QRS_NEXT_CUT()
PTP {E1 23936.911,E2 23936.911}
PTP {X 0,Y 607.929,A -85,B 0,C 180,E1 23936.911,E2 23936.911,E3 0,E4 0,E5 0,E6 0}
QRS_SPEED_INIT()
LIN {X 0,Y 607.929,Z 1180,A -85,B 0,C 180,E1 23936.911,E2 23936.911,E3 0,E4 0,E5 0,E6 0} C_VEL
LIN {X 0,Y 607.929,Z 517.391,A -85,B 0,C 180,E1 23936.911,E2 23936.911} C_VEL
LIN {X 0,Y 607.929,Z 509.316,A -85,B 0,C 180,E1 23936.911,E2 23936.911} C_VEL
LIN {X 0,Y 607.912,Z 507.316,A -85,B 0,C 180,E1 23936.722,E2 23936.722} C_VEL
LIN {X 0,Y 607.897,Z 507.324,A -85,B 0,C 180,E1 23933.441,E2 23933.441} C_VEL
LIN {X 0,Y 607.905,Z 507.318,A -85,B 0,C 180,E1 23930.246,E2 23930.246} C_VEL
LIN {X 0,Y 607.895,Z 507.323,A -85,B 0,C 180,E1 23927.074,E2 23927.074} C_VEL
LIN {X 0,Y 607.904,Z 507.318,A -85,B 0,C 180,E1 23923.861,E2 23923.861} C_VEL
LIN {X 0,Y 607.891,Z 507.323,A -85,B 0,C 180,E1 23920.694,E2 23920.694} C_VEL
LIN {X 0,Y 607.905,Z 507.318,A -85,B 0,C 180,E1 23917.568,E2 23917.568} C_VEL
LIN {X 0,Y 607.89,Z 507.323,A -85,B 0,C 180,E1 23914.337,E2 23914.337} C_VEL
LIN {X 0,Y 607.906,Z 507.318,A -85,B 0,C 180,E1 23911.189,E2 23911.189} C_VEL
LIN {X 0,Y 607.89,Z 507.324,A -85,B 0,C 180,E1 23908.02,E2 23908.02} C_VEL
LIN {X 0,Y 607.906,Z 507.318,A -85,B 0,C 180,E1 23904.83,E2 23904.83} C_VEL
LIN {X 0,Y 607.889,Z 507.324,A -85,B 0,C 180,E1 23901.677,E2 23901.677} C_VEL
LIN {X 0,Y 607.912,Z 507.317,A -85,B 0,C 180,E1 23898.591,E2 23898.591} C_VEL
LIN {X 0,Y 607.89,Z 507.324,A -85,B 0,C 180,E1 23895.386,E2 23895.386} C_VEL
LIN {X 0,Y 607.912,Z 507.315,A -85,B 0,C 180,E1 23892.257,E2 23892.257} C_VEL
LIN {X 0,Y 607.889,Z 507.318,A -85,B 0,C 180,E1 23889.047,E2 23889.047} C_VEL
LIN {X 0,Y 607.907,Z 507.606,A -85,B 0,C 180,E1 23887.52,E2 23887.52} C_VEL
LIN {X 0,Y 607.916,Z 514.249,A -85,B 0,C 180,E1 23887.05,E2 23887.05} C_VEL
LIN {X 0,Y 607.906,Z 561.512,A -85,B 0,C 180,E1 23884.062,E2 23884.062} C_VEL
LIN {X 0,Y 607.911,Z 589.892,A -85,B 0,C 180,E1 23882.327,E2 23882.327} C_VEL
LIN {X 0,Y 607.909,Z 810.334,A -85,B 0,C 180,E1 23879.35,E2 23879.35} C_VEL
LIN {X 0,Y 607.901,Z 895.692,A -85,B 0,C 180,E1 23878.194,E2 23878.194} C_VEL
LIN {X 0,Y 607.907,Z 916.51,A -85,B 0,C 180,E1 23877.74,E2 23877.74} C_VEL
LIN {X 0,Y 607.901,Z 936.743,A -85,B 0,C 180,E1 23877.149,E2 23877.149} C_VEL
LIN {X 0,Y 607.903,Z 957.25,A -85,B 0,C 180,E1 23876.365,E2 23876.365} C_VEL
LIN {X 0,Y 607.919,Z 978.375,A -85,B 0,C 180,E1 23875.369,E2 23875.369} C_VEL
LIN {X 0,Y 607.917,Z 997.713,A -85,B 0,C 180,E1 23874.279,E2 23874.279} C_VEL
LIN {X 0,Y 607.913,Z 1016.873,A -85,B 0,C 180,E1 23872.994,E2 23872.994} C_VEL
LIN {X 0,Y 607.911,Z 1034.44,A -85,B 0,C 180,E1 23871.618,E2 23871.618} C_VEL
LIN {X 0,Y 607.914,Z 1051.345,A -85,B 0,C 180,E1 23870.091,E2 23870.091} C_VEL
LIN {X 0,Y 607.918,Z 1066.577,A -85,B 0,C 180,E1 23868.508,E2 23868.508} C_VEL
LIN {X 0,Y 607.913,Z 1081.255,A -85,B 0,C 180,E1 23866.728,E2 23866.728} C_VEL
LIN {X 0,Y 607.918,Z 1093.745,A -85,B 0,C 180,E1 23864.965,E2 23864.965} C_VEL
LIN {X 0,Y 607.915,Z 1104.988,A -85,B 0,C 180,E1 23863.119,E2 23863.119} C_VEL
LIN {X 0,Y 607.902,Z 1114.343,A -85,B 0,C 180,E1 23861.287,E2 23861.287} C_VEL
LIN {X 0,Y 607.895,Z 1122.796,A -85,B 0,C 180,E1 23859.276,E2 23859.276} C_VEL
LIN {X 0,Y 607.892,Z 1129.344,A -85,B 0,C 180,E1 23857.336,E2 23857.336} C_VEL
LIN {X 0,Y 607.903,Z 1134.211,A -85,B 0,C 180,E1 23855.379,E2 23855.379} C_VEL
LIN {X 0,Y 607.918,Z 1137.791,A -85,B 0,C 180,E1 23853.291,E2 23853.291} C_VEL
LIN {X 0,Y 607.906,Z 1139.682,A -85,B 0,C 180,E1 23851.225,E2 23851.225} C_VEL
LIN {X 0,Y 607.894,Z 1139.839,A -85,B 0,C 180,E1 23849.246,E2 23849.246} C_VEL
LIN {X 0,Y 607.89,Z 1138.448,A -85,B 0,C 180,E1 23847.172,E2 23847.172} C_VEL
LIN {X 0,Y 607.898,Z 1135.562,A -85,B 0,C 180,E1 23845.188,E2 23845.188} C_VEL
LIN {X 0,Y 607.912,Z 1131.018,A -85,B 0,C 180,E1 23843.199,E2 23843.199} C_VEL
LIN {X 0,Y 607.914,Z 1124.904,A -85,B 0,C 180,E1 23841.201,E2 23841.201} C_VEL
LIN {X 0,Y 607.915,Z 1117.347,A -85,B 0,C 180,E1 23839.289,E2 23839.289} C_VEL
LIN {X 0,Y 607.919,Z 1107.548,A -85,B 0,C 180,E1 23837.268,E2 23837.268} C_VEL
LIN {X 0,Y 607.909,Z 1096.903,A -85,B 0,C 180,E1 23835.425,E2 23835.425} C_VEL
LIN {X 0,Y 607.904,Z 1084.856,A -85,B 0,C 180,E1 23833.665,E2 23833.665} C_VEL
LIN {X 0,Y 607.905,Z 1070.749,A -85,B 0,C 180,E1 23831.889,E2 23831.889} C_VEL
LIN {X 0,Y 607.907,Z 1055.655,A -85,B 0,C 180,E1 23830.245,E2 23830.245} C_VEL
LIN {X 0,Y 607.917,Z 1039.131,A -85,B 0,C 180,E1 23828.686,E2 23828.686} C_VEL
LIN {X 0,Y 607.915,Z 1021.54,A -85,B 0,C 180,E1 23827.262,E2 23827.262} C_VEL
LIN {X 0,Y 607.914,Z 1003.129,A -85,B 0,C 180,E1 23825.979,E2 23825.979} C_VEL
LIN {X 0,Y 607.918,Z 984.068,A -85,B 0,C 180,E1 23824.839,E2 23824.839} C_VEL
LIN {X 0,Y 607.899,Z 964.13,A -85,B 0,C 180,E1 23823.845,E2 23823.845} C_VEL
LIN {X 0,Y 607.905,Z 943.434,A -85,B 0,C 180,E1 23823.002,E2 23823.002} C_VEL
LIN {X 0,Y 607.919,Z 923.113,A -85,B 0,C 180,E1 23822.34,E2 23822.34} C_VEL
LIN {X 0,Y 607.899,Z 903.147,A -85,B 0,C 180,E1 23821.862,E2 23821.862} C_VEL
LIN {X 0,Y 607.912,Z 880.849,A -85,B 0,C 180,E1 23821.493,E2 23821.493} C_VEL
LIN {X 0,Y 607.908,Z 657.225,A -85,B 0,C 180,E1 23818.505,E2 23818.505} C_VEL
LIN {X 0,Y 607.879,Z 590.566,A -85,B 0,C 180,E1 23817.573,E2 23817.573} C_VEL
LIN {X 0,Y 607.88,Z 553.803,A -85,B 0,C 180,E1 23814.852,E2 23814.852} C_VEL
LIN {X 0,Y 607.917,Z 516.413,A -85,B 0,C 180,E1 23811.983,E2 23811.983} C_VEL
LIN {X 0,Y 607.886,Z 507.556,A -85,B 0,C 180,E1 23811.25,E2 23811.25} C_VEL
LIN {X 0,Y 607.85,Z 507.325,A -85,B 0,C 180,E1 23808.478,E2 23808.478} C_VEL
LIN {X 0,Y 607.917,Z 507.323,A -85,B 0,C 180,E1 23805.388,E2 23805.388} C_VEL
LIN {X 0,Y 607.847,Z 507.322,A -85,B 0,C 180,E1 23802.282,E2 23802.282} C_VEL
LIN {X 0,Y 607.891,Z 507.322,A -85,B 0,C 180,E1 23799.371,E2 23799.371} C_VEL
LIN {X 0,Y 607.853,Z 507.325,A -85,B 0,C 180,E1 23796.194,E2 23796.194} C_VEL
LIN {X 0,Y 607.85,Z 507.327,A -85,B 0,C 180,E1 23793.439,E2 23793.439} C_VEL
LIN {X 0,Y 607.919,Z 507.587,A -85,B 0,C 180,E1 23792.732,E2 23792.732} C_VEL
LIN {X 0,Y 607.906,Z 538.837,A -85,B 0,C 180,E1 23790.328,E2 23790.328} C_VEL
LIN {X 0,Y 607.862,Z 578.086,A -85,B 0,C 180,E1 23787.424,E2 23787.424} C_VEL
LIN {X 0,Y 607.911,Z 621.698,A -85,B 0,C 180,E1 23784.28,E2 23784.28} C_VEL
LIN {X 0,Y 607.876,Z 665.312,A -85,B 0,C 180,E1 23781.215,E2 23781.215} C_VEL
LIN {X 0,Y 607.877,Z 705.235,A -85,B 0,C 180,E1 23778.478,E2 23778.478} C_VEL
LIN {X 0,Y 607.916,Z 875.273,A -85,B 0,C 180,E1 23776.384,E2 23776.384} C_VEL
LIN {X 0,Y 607.919,Z 892.77,A -85,B 0,C 180,E1 23775.992,E2 23775.992} C_VEL
LIN {X 0,Y 607.902,Z 910.421,A -85,B 0,C 180,E1 23775.405,E2 23775.405} C_VEL
LIN {X 0,Y 607.901,Z 926.707,A -85,B 0,C 180,E1 23774.673,E2 23774.673} C_VEL
LIN {X 0,Y 607.92,Z 941.895,A -85,B 0,C 180,E1 23773.797,E2 23773.797} C_VEL
LIN {X 0,Y 607.919,Z 956.405,A -85,B 0,C 180,E1 23772.754,E2 23772.754} C_VEL
LIN {X 0,Y 607.918,Z 969.793,A -85,B 0,C 180,E1 23771.576,E2 23771.576} C_VEL
LIN {X 0,Y 607.916,Z 981.394,A -85,B 0,C 180,E1 23770.328,E2 23770.328} C_VEL
LIN {X 0,Y 607.914,Z 991.541,A -85,B 0,C 180,E1 23768.99,E2 23768.99} C_VEL
LIN {X 0,Y 607.916,Z 1000.812,A -85,B 0,C 180,E1 23767.466,E2 23767.466} C_VEL
LIN {X 0,Y 607.913,Z 1008.021,A -85,B 0,C 180,E1 23765.948,E2 23765.948} C_VEL
LIN {X 0,Y 607.913,Z 1013.696,A -85,B 0,C 180,E1 23764.339,E2 23764.339} C_VEL
LIN {X 0,Y 607.911,Z 1017.471,A -85,B 0,C 180,E1 23762.734,E2 23762.734} C_VEL
LIN {X 0,Y 607.919,Z 1019.517,A -85,B 0,C 180,E1 23761.131,E2 23761.131} C_VEL
LIN {X 0,Y 607.914,Z 1019.884,A -85,B 0,C 180,E1 23759.435,E2 23759.435} C_VEL
LIN {X 0,Y 607.909,Z 1018.533,A -85,B 0,C 180,E1 23757.832,E2 23757.832} C_VEL
LIN {X 0,Y 607.917,Z 1015.457,A -85,B 0,C 180,E1 23756.228,E2 23756.228} C_VEL
LIN {X 0,Y 607.917,Z 1010.558,A -85,B 0,C 180,E1 23754.621,E2 23754.621} C_VEL
LIN {X 0,Y 607.913,Z 1003.717,A -85,B 0,C 180,E1 23753.009,E2 23753.009} C_VEL
LIN {X 0,Y 607.915,Z 995.274,A -85,B 0,C 180,E1 23751.488,E2 23751.488} C_VEL
LIN {X 0,Y 607.914,Z 985.223,A -85,B 0,C 180,E1 23750.056,E2 23750.056} C_VEL
LIN {X 0,Y 607.914,Z 973.535,A -85,B 0,C 180,E1 23748.713,E2 23748.713} C_VEL
LIN {X 0,Y 607.919,Z 960.739,A -85,B 0,C 180,E1 23747.51,E2 23747.51} C_VEL
LIN {X 0,Y 607.92,Z 946.473,A -85,B 0,C 180,E1 23746.418,E2 23746.418} C_VEL
LIN {X 0,Y 607.899,Z 931.106,A -85,B 0,C 180,E1 23745.474,E2 23745.474} C_VEL
LIN {X 0,Y 607.908,Z 915.022,A -85,B 0,C 180,E1 23744.694,E2 23744.694} C_VEL
LIN {X 0,Y 607.919,Z 898.453,A -85,B 0,C 180,E1 23744.083,E2 23744.083} C_VEL
LIN {X 0,Y 607.92,Z 881.362,A -85,B 0,C 180,E1 23743.641,E2 23743.641} C_VEL
LIN {X 0,Y 607.896,Z 861.144,A -85,B 0,C 180,E1 23743.333,E2 23743.333} C_VEL
LIN {X 0,Y 607.875,Z 704.891,A -85,B 0,C 180,E1 23741.417,E2 23741.417} C_VEL
LIN {X 0,Y 607.886,Z 662.978,A -85,B 0,C 180,E1 23738.533,E2 23738.533} C_VEL
LIN {X 0,Y 607.904,Z 617.88,A -85,B 0,C 180,E1 23735.358,E2 23735.358} C_VEL
LIN {X 0,Y 607.863,Z 576.988,A -85,B 0,C 180,E1 23732.406,E2 23732.406} C_VEL
LIN {X 0,Y 607.918,Z 536.407,A -85,B 0,C 180,E1 23729.4,E2 23729.4} C_VEL
LIN {X 0,Y 607.917,Z 507.644,A -85,B 0,C 180,E1 23727.189,E2 23727.189} C_VEL
LIN {X 0,Y 607.846,Z 507.328,A -85,B 0,C 180,E1 23726.335,E2 23726.335} C_VEL
LIN {X 0,Y 607.917,Z 507.326,A -85,B 0,C 180,E1 23723.342,E2 23723.342} C_VEL
LIN {X 0,Y 607.881,Z 507.321,A -85,B 0,C 180,E1 23720.187,E2 23720.187} C_VEL
LIN {X 0,Y 607.898,Z 507.322,A -85,B 0,C 180,E1 23717.083,E2 23717.083} C_VEL
LIN {X 0,Y 607.907,Z 507.325,A -85,B 0,C 180,E1 23713.913,E2 23713.913} C_VEL
LIN {X 0,Y 607.871,Z 507.312,A -85,B 0,C 180,E1 23710.832,E2 23710.832} C_VEL
LIN {X 0,Y 607.915,Z 507.658,A -85,B 0,C 180,E1 23709.994,E2 23709.994} C_VEL
LIN {X 0,Y 607.916,Z 539.976,A -85,B 0,C 180,E1 23707.604,E2 23707.604} C_VEL
LIN {X 0,Y 607.912,Z 544.123,A -85,B 0,C 180,E1 23707.352,E2 23707.352} C_VEL
LIN {X 0,Y 607.919,Z 747.532,A -85,B 0,C 180,E1 23704.443,E2 23704.443} C_VEL
LIN {X 0,Y 607.913,Z 889.955,A -85,B 0,C 180,E1 23702.443,E2 23702.443} C_VEL
LIN {X 0,Y 607.918,Z 912.241,A -85,B 0,C 180,E1 23701.979,E2 23701.979} C_VEL
LIN {X 0,Y 607.918,Z 931.576,A -85,B 0,C 180,E1 23701.425,E2 23701.425} C_VEL
LIN {X 0,Y 607.913,Z 951.698,A -85,B 0,C 180,E1 23700.713,E2 23700.713} C_VEL
LIN {X 0,Y 607.918,Z 972.94,A -85,B 0,C 180,E1 23699.783,E2 23699.783} C_VEL
LIN {X 0,Y 607.916,Z 992.693,A -85,B 0,C 180,E1 23698.761,E2 23698.761} C_VEL
LIN {X 0,Y 607.918,Z 1012.955,A -85,B 0,C 180,E1 23697.527,E2 23697.527} C_VEL
LIN {X 0,Y 607.915,Z 1031.87,A -85,B 0,C 180,E1 23696.207,E2 23696.207} C_VEL
LIN {X 0,Y 607.917,Z 1050.602,A -85,B 0,C 180,E1 23694.693,E2 23694.693} C_VEL
LIN {X 0,Y 607.914,Z 1068.568,A -85,B 0,C 180,E1 23693.045,E2 23693.045} C_VEL
LIN {X 0,Y 607.918,Z 1085.053,A -85,B 0,C 180,E1 23691.314,E2 23691.314} C_VEL
LIN {X 0,Y 607.911,Z 1100.102,A -85,B 0,C 180,E1 23689.505,E2 23689.505} C_VEL
LIN {X 0,Y 607.901,Z 1113.944,A -85,B 0,C 180,E1 23687.616,E2 23687.616} C_VEL
LIN {X 0,Y 607.89,Z 1125.712,A -85,B 0,C 180,E1 23685.747,E2 23685.747} C_VEL
LIN {X 0,Y 607.905,Z 1136.434,A -85,B 0,C 180,E1 23683.798,E2 23683.798} C_VEL
LIN {X 0,Y 607.894,Z 1145.337,A -85,B 0,C 180,E1 23681.863,E2 23681.863} C_VEL
LIN {X 0,Y 607.886,Z 1153.183,A -85,B 0,C 180,E1 23679.85,E2 23679.85} C_VEL
LIN {X 0,Y 607.916,Z 1159.569,A -85,B 0,C 180,E1 23677.751,E2 23677.751} C_VEL
LIN {X 0,Y 607.888,Z 1164.493,A -85,B 0,C 180,E1 23675.664,E2 23675.664} C_VEL
LIN {X 0,Y 607.894,Z 1167.728,A -85,B 0,C 180,E1 23673.583,E2 23673.583} C_VEL
LIN {X 0,Y 607.907,Z 1169.591,A -85,B 0,C 180,E1 23671.508,E2 23671.508} C_VEL
LIN {X 0,Y 607.883,Z 1169.872,A -85,B 0,C 180,E1 23669.435,E2 23669.435} C_VEL
LIN {X 0,Y 607.919,Z 1168.853,A -85,B 0,C 180,E1 23667.455,E2 23667.455} C_VEL
LIN {X 0,Y 607.899,Z 1166.116,A -85,B 0,C 180,E1 23665.283,E2 23665.283} C_VEL
LIN {X 0,Y 607.895,Z 1162.22,A -85,B 0,C 180,E1 23663.294,E2 23663.294} C_VEL
LIN {X 0,Y 607.914,Z 1156.257,A -85,B 0,C 180,E1 23661.106,E2 23661.106} C_VEL
LIN {X 0,Y 607.901,Z 1149.266,A -85,B 0,C 180,E1 23659.097,E2 23659.097} C_VEL
LIN {X 0,Y 607.895,Z 1140.146,A -85,B 0,C 180,E1 23656.977,E2 23656.977} C_VEL
LIN {X 0,Y 607.919,Z 1130.748,A -85,B 0,C 180,E1 23655.133,E2 23655.133} C_VEL
LIN {X 0,Y 607.915,Z 1118.445,A -85,B 0,C 180,E1 23653.075,E2 23653.075} C_VEL
LIN {X 0,Y 607.911,Z 1105.489,A -85,B 0,C 180,E1 23651.194,E2 23651.194} C_VEL
LIN {X 0,Y 607.907,Z 1090.93,A -85,B 0,C 180,E1 23649.367,E2 23649.367} C_VEL
LIN {X 0,Y 607.906,Z 1074.652,A -85,B 0,C 180,E1 23647.568,E2 23647.568} C_VEL
LIN {X 0,Y 607.911,Z 1057.689,A -85,B 0,C 180,E1 23645.927,E2 23645.927} C_VEL
LIN {X 0,Y 607.912,Z 1039.251,A -85,B 0,C 180,E1 23644.369,E2 23644.369} C_VEL
LIN {X 0,Y 607.912,Z 1020.177,A -85,B 0,C 180,E1 23642.95,E2 23642.95} C_VEL
LIN {X 0,Y 607.915,Z 1000.251,A -85,B 0,C 180,E1 23641.68,E2 23641.68} C_VEL
LIN {X 0,Y 607.919,Z 978.842,A -85,B 0,C 180,E1 23640.504,E2 23640.504} C_VEL
LIN {X 0,Y 607.915,Z 959.663,A -85,B 0,C 180,E1 23639.618,E2 23639.618} C_VEL
LIN {X 0,Y 607.912,Z 938.247,A -85,B 0,C 180,E1 23638.788,E2 23638.788} C_VEL
LIN {X 0,Y 607.915,Z 917.429,A -85,B 0,C 180,E1 23638.16,E2 23638.16} C_VEL
LIN {X 0,Y 607.91,Z 895.972,A -85,B 0,C 180,E1 23637.659,E2 23637.659} C_VEL
LIN {X 0,Y 607.913,Z 861.646,A -85,B 0,C 180,E1 23637.143,E2 23637.143} C_VEL
LIN {X 0,Y 607.918,Z 650.979,A -85,B 0,C 180,E1 23634.191,E2 23634.191} C_VEL
LIN {X 0,Y 607.918,Z 541.954,A -85,B 0,C 180,E1 23632.598,E2 23632.598} C_VEL
LIN {X 0,Y 607.903,Z 507.829,A -85,B 0,C 180,E1 23630.506,E2 23630.506} C_VEL
LIN {X 0,Y 607.898,Z 507.371,A -85,B 0,C 180,E1 23630.332,E2 23630.332} C_VEL
LIN {X 0,Y 607.891,Z 507.319,A -85,B 0,C 180,E1 23627.211,E2 23627.211} C_VEL
LIN {X 0,Y 607.901,Z 507.324,A -85,B 0,C 180,E1 23624.086,E2 23624.086} C_VEL
LIN {X 0,Y 607.896,Z 507.318,A -85,B 0,C 180,E1 23620.978,E2 23620.978} C_VEL
LIN {X 0,Y 607.904,Z 507.324,A -85,B 0,C 180,E1 23617.842,E2 23617.842} C_VEL
LIN {X 0,Y 607.899,Z 507.318,A -85,B 0,C 180,E1 23614.675,E2 23614.675} C_VEL
LIN {X 0,Y 607.905,Z 507.325,A -85,B 0,C 180,E1 23611.536,E2 23611.536} C_VEL
LIN {X 0,Y 607.902,Z 507.317,A -85,B 0,C 180,E1 23608.363,E2 23608.363} C_VEL
LIN {X 0,Y 607.905,Z 507.325,A -85,B 0,C 180,E1 23605.213,E2 23605.213} C_VEL
LIN {X 0,Y 607.903,Z 507.316,A -85,B 0,C 180,E1 23602.024,E2 23602.024} C_VEL
LIN {X 0,Y 607.901,Z 507.324,A -85,B 0,C 180,E1 23598.806,E2 23598.806} C_VEL
LIN {X 0,Y 607.902,Z 507.316,A -85,B 0,C 180,E1 23595.649,E2 23595.649} C_VEL
LIN {X 0,Y 607.898,Z 507.324,A -85,B 0,C 180,E1 23592.443,E2 23592.443} C_VEL
LIN {X 0,Y 607.902,Z 507.317,A -85,B 0,C 180,E1 23589.276,E2 23589.276} C_VEL
LIN {X 0,Y 607.9,Z 507.324,A -85,B 0,C 180,E1 23586.137,E2 23586.137} C_VEL
LIN {X 0,Y 607.902,Z 507.318,A -85,B 0,C 180,E1 23582.922,E2 23582.922} C_VEL
LIN {X 0,Y 607.895,Z 507.323,A -85,B 0,C 180,E1 23579.717,E2 23579.717} C_VEL
LIN {X 0,Y 607.912,Z 507.316,A -85,B 0,C 180,E1 23576.722,E2 23576.722} C_VEL
LIN {X 0,Y 606.898,Z 507.452,A -85,B 0,C 180,E1 23575.996,E2 23575.996} C_VEL
LIN {X 0,Y 600.503,Z 508.251,A -85,B 0,C 180,E1 23573.959,E2 23573.959} C_VEL
LIN {X 0,Y 599.958,Z 508.312,A -85,B 0,C 180,E1 23573.429,E2 23573.429} C_VEL
LIN {X 0,Y 599.965,Z 508.307,A -85,B 0,C 180,E1 23570.213,E2 23570.213} C_VEL
LIN {X 0,Y 599.953,Z 508.31,A -85,B 0,C 180,E1 23566.998,E2 23566.998} C_VEL
LIN {X 0,Y 599.964,Z 508.308,A -85,B 0,C 180,E1 23563.84,E2 23563.84} C_VEL
LIN {X 0,Y 599.95,Z 508.31,A -85,B 0,C 180,E1 23560.631,E2 23560.631} C_VEL
LIN {X 0,Y 599.962,Z 508.308,A -85,B 0,C 180,E1 23557.461,E2 23557.461} C_VEL
LIN {X 0,Y 599.951,Z 508.311,A -85,B 0,C 180,E1 23554.322,E2 23554.322} C_VEL
LIN {X 0,Y 599.968,Z 508.307,A -85,B 0,C 180,E1 23551.208,E2 23551.208} C_VEL
LIN {X 0,Y 599.951,Z 508.312,A -85,B 0,C 180,E1 23547.996,E2 23547.996} C_VEL
LIN {X 0,Y 599.966,Z 508.307,A -85,B 0,C 180,E1 23544.787,E2 23544.787} C_VEL
LIN {X 0,Y 599.951,Z 508.313,A -85,B 0,C 180,E1 23541.686,E2 23541.686} C_VEL
LIN {X 0,Y 599.973,Z 508.306,A -85,B 0,C 180,E1 23538.578,E2 23538.578} C_VEL
LIN {X 0,Y 599.951,Z 508.314,A -85,B 0,C 180,E1 23535.368,E2 23535.368} C_VEL
LIN {X 0,Y 599.97,Z 508.304,A -85,B 0,C 180,E1 23532.191,E2 23532.191} C_VEL
LIN {X 0,Y 599.949,Z 508.299,A -85,B 0,C 180,E1 23529.047,E2 23529.047} C_VEL
LIN {X 0,Y 600.017,Z 508.588,A -85,B 0,C 180,E1 23528.035,E2 23528.035} C_VEL
LIN {X 0,Y 601.153,Z 512.117,A -85,B 0,C 180,E1 23527.679,E2 23527.679} C_VEL
LIN {X 0,Y 600.962,Z 558.146,A -85,B 0,C 180,E1 23524.724,E2 23524.724} C_VEL
LIN {X 0,Y 600.962,Z 590.28,A -85,B 0,C 180,E1 23522.74,E2 23522.74} C_VEL
LIN {X 0,Y 601,Z 716.679,A -85,B 0,C 180,E1 23520.992,E2 23520.992} C_VEL
LIN {X 0,Y 600.845,Z 895.307,A -85,B 0,C 180,E1 23518.562,E2 23518.562} C_VEL
LIN {X 0,Y 600.787,Z 916.41,A -85,B 0,C 180,E1 23518.102,E2 23518.102} C_VEL
LIN {X 0,Y 600.703,Z 937.346,A -85,B 0,C 180,E1 23517.48,E2 23517.48} C_VEL
LIN {X 0,Y 600.635,Z 957.269,A -85,B 0,C 180,E1 23516.709,E2 23516.709} C_VEL
LIN {X 0,Y 600.54,Z 978.39,A -85,B 0,C 180,E1 23515.704,E2 23515.704} C_VEL
LIN {X 0,Y 600.445,Z 997.721,A -85,B 0,C 180,E1 23514.601,E2 23514.601} C_VEL
LIN {X 0,Y 600.351,Z 1016.885,A -85,B 0,C 180,E1 23513.3,E2 23513.3} C_VEL
LIN {X 0,Y 600.247,Z 1034.524,A -85,B 0,C 180,E1 23511.902,E2 23511.902} C_VEL
LIN {X 0,Y 600.158,Z 1051.207,A -85,B 0,C 180,E1 23510.377,E2 23510.377} C_VEL
LIN {X 0,Y 600.103,Z 1066.583,A -85,B 0,C 180,E1 23508.758,E2 23508.758} C_VEL
LIN {X 0,Y 600.045,Z 1081.261,A -85,B 0,C 180,E1 23506.954,E2 23506.954} C_VEL
LIN {X 0,Y 599.995,Z 1093.751,A -85,B 0,C 180,E1 23505.167,E2 23505.167} C_VEL
LIN {X 0,Y 599.955,Z 1105.093,A -85,B 0,C 180,E1 23503.277,E2 23503.277} C_VEL
LIN {X 0,Y 599.925,Z 1114.347,A -85,B 0,C 180,E1 23501.439,E2 23501.439} C_VEL
LIN {X 0,Y 599.905,Z 1122.798,A -85,B 0,C 180,E1 23499.401,E2 23499.401} C_VEL
LIN {X 0,Y 599.901,Z 1129.243,A -85,B 0,C 180,E1 23497.47,E2 23497.47} C_VEL
LIN {X 0,Y 599.909,Z 1134.212,A -85,B 0,C 180,E1 23495.451,E2 23495.451} C_VEL
LIN {X 0,Y 599.917,Z 1137.821,A -85,B 0,C 180,E1 23493.311,E2 23493.311} C_VEL
LIN {X 0,Y 599.906,Z 1139.683,A -85,B 0,C 180,E1 23491.242,E2 23491.242} C_VEL
LIN {X 0,Y 599.894,Z 1139.839,A -85,B 0,C 180,E1 23489.236,E2 23489.236} C_VEL
LIN {X 0,Y 599.891,Z 1138.448,A -85,B 0,C 180,E1 23487.134,E2 23487.134} C_VEL
LIN {X 0,Y 599.895,Z 1135.561,A -85,B 0,C 180,E1 23485.124,E2 23485.124} C_VEL
LIN {X 0,Y 599.913,Z 1131.017,A -85,B 0,C 180,E1 23483.108,E2 23483.108} C_VEL
LIN {X 0,Y 599.927,Z 1124.903,A -85,B 0,C 180,E1 23481.083,E2 23481.083} C_VEL
LIN {X 0,Y 599.933,Z 1117.345,A -85,B 0,C 180,E1 23479.145,E2 23479.145} C_VEL
LIN {X 0,Y 599.957,Z 1107.546,A -85,B 0,C 180,E1 23477.096,E2 23477.096} C_VEL
LIN {X 0,Y 599.988,Z 1096.898,A -85,B 0,C 180,E1 23475.228,E2 23475.228} C_VEL
LIN {X 0,Y 600.012,Z 1084.339,A -85,B 0,C 180,E1 23473.371,E2 23473.371} C_VEL
LIN {X 0,Y 600.073,Z 1070.745,A -85,B 0,C 180,E1 23471.644,E2 23471.644} C_VEL
LIN {X 0,Y 600.152,Z 1055.142,A -85,B 0,C 180,E1 23469.928,E2 23469.928} C_VEL
LIN {X 0,Y 600.243,Z 1038.618,A -85,B 0,C 180,E1 23468.356,E2 23468.356} C_VEL
LIN {X 0,Y 600.313,Z 1020.872,A -85,B 0,C 180,E1 23466.906,E2 23466.906} C_VEL
LIN {X 0,Y 600.419,Z 1002.319,A -85,B 0,C 180,E1 23465.607,E2 23465.607} C_VEL
LIN {X 0,Y 600.528,Z 983.065,A -85,B 0,C 180,E1 23464.454,E2 23464.454} C_VEL
LIN {X 0,Y 600.585,Z 964.12,A -85,B 0,C 180,E1 23463.502,E2 23463.502} C_VEL
LIN {X 0,Y 600.69,Z 943.418,A -85,B 0,C 180,E1 23462.651,E2 23462.651} C_VEL
LIN {X 0,Y 600.787,Z 922.72,A -85,B 0,C 180,E1 23461.973,E2 23461.973} C_VEL
LIN {X 0,Y 600.819,Z 902.146,A -85,B 0,C 180,E1 23461.48,E2 23461.48} C_VEL
LIN {X 0,Y 600.887,Z 875.462,A -85,B 0,C 180,E1 23461.057,E2 23461.057} C_VEL
LIN {X 0,Y 601.1,Z 646.863,A -85,B 0,C 180,E1 23457.965,E2 23457.965} C_VEL
LIN {X 0,Y 600.943,Z 591.711,A -85,B 0,C 180,E1 23457.186,E2 23457.186} C_VEL
LIN {X 0,Y 600.756,Z 588.796,A -85,B 0,C 180,E1 23457.016,E2 23457.016} C_VEL
LIN {X 0,Y 600.905,Z 549.973,A -85,B 0,C 180,E1 23454.089,E2 23454.089} C_VEL
LIN {X 0,Y 601.087,Z 512.529,A -85,B 0,C 180,E1 23451.163,E2 23451.163} C_VEL
LIN {X 0,Y 600.742,Z 510.965,A -85,B 0,C 180,E1 23451.011,E2 23451.011} C_VEL
LIN {X 0,Y 599.935,Z 508.477,A -85,B 0,C 180,E1 23450.705,E2 23450.705} C_VEL
LIN {X 0,Y 599.957,Z 508.313,A -85,B 0,C 180,E1 23447.807,E2 23447.807} C_VEL
LIN {X 0,Y 599.915,Z 508.315,A -85,B 0,C 180,E1 23444.561,E2 23444.561} C_VEL
LIN {X 0,Y 599.93,Z 508.306,A -85,B 0,C 180,E1 23441.681,E2 23441.681} C_VEL
LIN {X 0,Y 599.925,Z 508.315,A -85,B 0,C 180,E1 23438.434,E2 23438.434} C_VEL
LIN {X 0,Y 599.912,Z 508.312,A -85,B 0,C 180,E1 23435.568,E2 23435.568} C_VEL
LIN {X 0,Y 599.961,Z 508.511,A -85,B 0,C 180,E1 23433.16,E2 23433.16} C_VEL
LIN {X 0,Y 600.756,Z 511.229,A -85,B 0,C 180,E1 23432.859,E2 23432.859} C_VEL
LIN {X 0,Y 600.558,Z 549.022,A -85,B 0,C 180,E1 23429.965,E2 23429.965} C_VEL
LIN {X 0,Y 600.493,Z 588.443,A -85,B 0,C 180,E1 23427.024,E2 23427.024} C_VEL
LIN {X 0,Y 600.358,Z 631.884,A -85,B 0,C 180,E1 23423.873,E2 23423.873} C_VEL
LIN {X 0,Y 600.22,Z 674.045,A -85,B 0,C 180,E1 23420.885,E2 23420.885} C_VEL
LIN {X 0,Y 600.219,Z 705.587,A -85,B 0,C 180,E1 23418.714,E2 23418.714} C_VEL
LIN {X 0,Y 600.236,Z 875.808,A -85,B 0,C 180,E1 23416.59,E2 23416.59} C_VEL
LIN {X 0,Y 600.209,Z 893.333,A -85,B 0,C 180,E1 23416.187,E2 23416.187} C_VEL
LIN {X 0,Y 600.157,Z 910.443,A -85,B 0,C 180,E1 23415.609,E2 23415.609} C_VEL
LIN {X 0,Y 600.115,Z 926.725,A -85,B 0,C 180,E1 23414.868,E2 23414.868} C_VEL
LIN {X 0,Y 600.082,Z 941.908,A -85,B 0,C 180,E1 23413.981,E2 23413.981} C_VEL
LIN {X 0,Y 600.038,Z 956.69,A -85,B 0,C 180,E1 23412.902,E2 23412.902} C_VEL
LIN {X 0,Y 600.002,Z 970.308,A -85,B 0,C 180,E1 23411.682,E2 23411.682} C_VEL
LIN {X 0,Y 599.965,Z 982.175,A -85,B 0,C 180,E1 23410.369,E2 23410.369} C_VEL
LIN {X 0,Y 599.943,Z 992.824,A -85,B 0,C 180,E1 23408.917,E2 23408.917} C_VEL
LIN {X 0,Y 599.932,Z 1001.644,A -85,B 0,C 180,E1 23407.412,E2 23407.412} C_VEL
LIN {X 0,Y 599.917,Z 1008.813,A -85,B 0,C 180,E1 23405.835,E2 23405.835} C_VEL
LIN {X 0,Y 599.915,Z 1014.209,A -85,B 0,C 180,E1 23404.206,E2 23404.206} C_VEL
LIN {X 0,Y 599.913,Z 1017.788,A -85,B 0,C 180,E1 23402.579,E2 23402.579} C_VEL
LIN {X 0,Y 599.913,Z 1019.719,A -85,B 0,C 180,E1 23400.86,E2 23400.86} C_VEL
LIN {X 0,Y 599.916,Z 1019.827,A -85,B 0,C 180,E1 23399.236,E2 23399.236} C_VEL
LIN {X 0,Y 599.911,Z 1018.25,A -85,B 0,C 180,E1 23397.612,E2 23397.612} C_VEL
LIN {X 0,Y 599.912,Z 1014.953,A -85,B 0,C 180,E1 23395.986,E2 23395.986} C_VEL
LIN {X 0,Y 599.921,Z 1009.848,A -85,B 0,C 180,E1 23394.357,E2 23394.357} C_VEL
LIN {X 0,Y 599.924,Z 1003.256,A -85,B 0,C 180,E1 23392.82,E2 23392.82} C_VEL
LIN {X 0,Y 599.938,Z 994.683,A -85,B 0,C 180,E1 23391.277,E2 23391.277} C_VEL
LIN {X 0,Y 599.959,Z 985.22,A -85,B 0,C 180,E1 23389.922,E2 23389.922} C_VEL
LIN {X 0,Y 599.988,Z 973.533,A -85,B 0,C 180,E1 23388.562,E2 23388.562} C_VEL
LIN {X 0,Y 600.026,Z 960.734,A -85,B 0,C 180,E1 23387.343,E2 23387.343} C_VEL
LIN {X 0,Y 600.073,Z 946.928,A -85,B 0,C 180,E1 23386.268,E2 23386.268} C_VEL
LIN {X 0,Y 600.095,Z 930.963,A -85,B 0,C 180,E1 23385.273,E2 23385.273} C_VEL
LIN {X 0,Y 600.144,Z 914.998,A -85,B 0,C 180,E1 23384.491,E2 23384.491} C_VEL
LIN {X 0,Y 600.2,Z 898.44,A -85,B 0,C 180,E1 23383.872,E2 23383.872} C_VEL
LIN {X 0,Y 600.235,Z 881.021,A -85,B 0,C 180,E1 23383.419,E2 23383.419} C_VEL
LIN {X 0,Y 600.229,Z 859.947,A -85,B 0,C 180,E1 23383.1,E2 23383.1} C_VEL
LIN {X 0,Y 600.175,Z 705.121,A -85,B 0,C 180,E1 23381.182,E2 23381.182} C_VEL
LIN {X 0,Y 600.279,Z 662.242,A -85,B 0,C 180,E1 23378.196,E2 23378.196} C_VEL
LIN {X 0,Y 600.396,Z 617.871,A -85,B 0,C 180,E1 23375.029,E2 23375.029} C_VEL
LIN {X 0,Y 600.473,Z 577.862,A -85,B 0,C 180,E1 23372.102,E2 23372.102} C_VEL
LIN {X 0,Y 600.665,Z 537.124,A -85,B 0,C 180,E1 23369.046,E2 23369.046} C_VEL
LIN {X 0,Y 600.723,Z 510.879,A -85,B 0,C 180,E1 23367.022,E2 23367.022} C_VEL
LIN {X 0,Y 599.954,Z 508.513,A -85,B 0,C 180,E1 23366.75,E2 23366.75} C_VEL
LIN {X 0,Y 599.936,Z 508.316,A -85,B 0,C 180,E1 23363.845,E2 23363.845} C_VEL
LIN {X 0,Y 599.952,Z 508.306,A -85,B 0,C 180,E1 23360.5,E2 23360.5} C_VEL
LIN {X 0,Y 599.963,Z 508.313,A -85,B 0,C 180,E1 23357.303,E2 23357.303} C_VEL
LIN {X 0,Y 599.967,Z 508.312,A -85,B 0,C 180,E1 23354.089,E2 23354.089} C_VEL
LIN {X 0,Y 599.929,Z 508.287,A -85,B 0,C 180,E1 23350.977,E2 23350.977} C_VEL
LIN {X 0,Y 600.006,Z 508.691,A -85,B 0,C 180,E1 23350.547,E2 23350.547} C_VEL
LIN {X 0,Y 601.227,Z 511.885,A -85,B 0,C 180,E1 23350.185,E2 23350.185} C_VEL
LIN {X 0,Y 601.152,Z 543.472,A -85,B 0,C 180,E1 23347.86,E2 23347.86} C_VEL
LIN {X 0,Y 601.539,Z 547.034,A -85,B 0,C 180,E1 23347.771,E2 23347.771} C_VEL
LIN {X 0,Y 601.308,Z 754.795,A -85,B 0,C 180,E1 23344.773,E2 23344.773} C_VEL
LIN {X 0,Y 601.147,Z 891.224,A -85,B 0,C 180,E1 23342.833,E2 23342.833} C_VEL
LIN {X 0,Y 601.07,Z 914.902,A -85,B 0,C 180,E1 23342.315,E2 23342.315} C_VEL
LIN {X 0,Y 601,Z 934.455,A -85,B 0,C 180,E1 23341.735,E2 23341.735} C_VEL
LIN {X 0,Y 600.876,Z 957.248,A -85,B 0,C 180,E1 23340.881,E2 23340.881} C_VEL
LIN {X 0,Y 600.793,Z 976.298,A -85,B 0,C 180,E1 23340.007,E2 23340.007} C_VEL
LIN {X 0,Y 600.656,Z 997.467,A -85,B 0,C 180,E1 23338.865,E2 23338.865} C_VEL
LIN {X 0,Y 600.556,Z 1016.891,A -85,B 0,C 180,E1 23337.63,E2 23337.63} C_VEL
LIN {X 0,Y 600.418,Z 1036.953,A -85,B 0,C 180,E1 23336.159,E2 23336.159} C_VEL
LIN {X 0,Y 600.324,Z 1055.725,A -85,B 0,C 180,E1 23334.581,E2 23334.581} C_VEL
LIN {X 0,Y 600.213,Z 1073.063,A -85,B 0,C 180,E1 23332.898,E2 23332.898} C_VEL
LIN {X 0,Y 600.124,Z 1090.283,A -85,B 0,C 180,E1 23330.99,E2 23330.99} C_VEL
LIN {X 0,Y 600.076,Z 1104.956,A -85,B 0,C 180,E1 23329.137,E2 23329.137} C_VEL
LIN {X 0,Y 600.019,Z 1118.447,A -85,B 0,C 180,E1 23327.155,E2 23327.155} C_VEL
LIN {X 0,Y 599.976,Z 1130.749,A -85,B 0,C 180,E1 23325.069,E2 23325.069} C_VEL
LIN {X 0,Y 599.925,Z 1140.147,A -85,B 0,C 180,E1 23323.199,E2 23323.199} C_VEL
LIN {X 0,Y 599.916,Z 1149.483,A -85,B 0,C 180,E1 23320.991,E2 23320.991} C_VEL
LIN {X 0,Y 599.925,Z 1156.257,A -85,B 0,C 180,E1 23319.013,E2 23319.013} C_VEL
LIN {X 0,Y 599.892,Z 1162.22,A -85,B 0,C 180,E1 23316.796,E2 23316.796} C_VEL
LIN {X 0,Y 599.902,Z 1166.116,A -85,B 0,C 180,E1 23314.78,E2 23314.78} C_VEL
LIN {X 0,Y 599.916,Z 1168.853,A -85,B 0,C 180,E1 23312.579,E2 23312.579} C_VEL
LIN {X 0,Y 599.883,Z 1169.872,A -85,B 0,C 180,E1 23310.573,E2 23310.573} C_VEL
LIN {X 0,Y 599.904,Z 1169.524,A -85,B 0,C 180,E1 23308.376,E2 23308.376} C_VEL
LIN {X 0,Y 599.897,Z 1167.728,A -85,B 0,C 180,E1 23306.369,E2 23306.369} C_VEL
LIN {X 0,Y 599.889,Z 1164.493,A -85,B 0,C 180,E1 23304.261,E2 23304.261} C_VEL
LIN {X 0,Y 599.916,Z 1159.57,A -85,B 0,C 180,E1 23302.145,E2 23302.145} C_VEL
LIN {X 0,Y 599.905,Z 1153.183,A -85,B 0,C 180,E1 23300.018,E2 23300.018} C_VEL
LIN {X 0,Y 599.914,Z 1145.33,A -85,B 0,C 180,E1 23297.975,E2 23297.975} C_VEL
LIN {X 0,Y 599.962,Z 1135.914,A -85,B 0,C 180,E1 23295.91,E2 23295.91} C_VEL
LIN {X 0,Y 599.977,Z 1125.133,A -85,B 0,C 180,E1 23293.94,E2 23293.94} C_VEL
LIN {X 0,Y 600.024,Z 1112.579,A -85,B 0,C 180,E1 23291.944,E2 23291.944} C_VEL
LIN {X 0,Y 600.076,Z 1099.326,A -85,B 0,C 180,E1 23290.129,E2 23290.129} C_VEL
LIN {X 0,Y 600.16,Z 1083.194,A -85,B 0,C 180,E1 23288.191,E2 23288.191} C_VEL
LIN {X 0,Y 600.271,Z 1066.529,A -85,B 0,C 180,E1 23286.437,E2 23286.437} C_VEL
LIN {X 0,Y 600.349,Z 1048.792,A -85,B 0,C 180,E1 23284.816,E2 23284.816} C_VEL
LIN {X 0,Y 600.479,Z 1028.385,A -85,B 0,C 180,E1 23283.187,E2 23283.187} C_VEL
LIN {X 0,Y 600.599,Z 1008.934,A -85,B 0,C 180,E1 23281.838,E2 23281.838} C_VEL
LIN {X 0,Y 600.716,Z 988.809,A -85,B 0,C 180,E1 23280.648,E2 23280.648} C_VEL
LIN {X 0,Y 600.843,Z 967.729,A -85,B 0,C 180,E1 23279.575,E2 23279.575} C_VEL
LIN {X 0,Y 600.941,Z 946.656,A -85,B 0,C 180,E1 23278.699,E2 23278.699} C_VEL
LIN {X 0,Y 601.031,Z 925.505,A -85,B 0,C 180,E1 23277.975,E2 23277.975} C_VEL
LIN {X 0,Y 601.109,Z 903.426,A -85,B 0,C 180,E1 23277.41,E2 23277.41} C_VEL
LIN {X 0,Y 601.158,Z 883.629,A -85,B 0,C 180,E1 23277.041,E2 23277.041} C_VEL
LIN {X 0,Y 601.403,Z 664.197,A -85,B 0,C 180,E1 23273.933,E2 23273.933} C_VEL
LIN {X 0,Y 601.379,Z 543.241,A -85,B 0,C 180,E1 23272.161,E2 23272.161} C_VEL
LIN {X 0,Y 601.249,Z 533.59,A -85,B 0,C 180,E1 23271.602,E2 23271.602} C_VEL
LIN {X 0,Y 601.325,Z 511.91,A -85,B 0,C 180,E1 23270.266,E2 23270.266} C_VEL
LIN {X 0,Y 600.002,Z 508.541,A -85,B 0,C 180,E1 23269.896,E2 23269.896} C_VEL
LIN {X 0,Y 599.955,Z 508.31,A -85,B 0,C 180,E1 23266.882,E2 23266.882} C_VEL
LIN {X 0,Y 599.964,Z 508.308,A -85,B 0,C 180,E1 23263.674,E2 23263.674} C_VEL
LIN {X 0,Y 599.956,Z 508.311,A -85,B 0,C 180,E1 23260.538,E2 23260.538} C_VEL
LIN {X 0,Y 599.962,Z 508.305,A -85,B 0,C 180,E1 23257.345,E2 23257.345} C_VEL
LIN {X 0,Y 599.958,Z 508.313,A -85,B 0,C 180,E1 23254.168,E2 23254.168} C_VEL
LIN {X 0,Y 599.962,Z 508.307,A -85,B 0,C 180,E1 23250.994,E2 23250.994} C_VEL
LIN {X 0,Y 599.962,Z 508.313,A -85,B 0,C 180,E1 23247.756,E2 23247.756} C_VEL
LIN {X 0,Y 599.969,Z 508.306,A -85,B 0,C 180,E1 23244.505,E2 23244.505} C_VEL
LIN {X 0,Y 599.972,Z 508.313,A -85,B 0,C 180,E1 23241.2,E2 23241.2} C_VEL
LIN {X 0,Y 599.968,Z 508.306,A -85,B 0,C 180,E1 23237.857,E2 23237.857} C_VEL
LIN {X 0,Y 599.966,Z 508.313,A -85,B 0,C 180,E1 23234.673,E2 23234.673} C_VEL
LIN {X 0,Y 599.965,Z 508.306,A -85,B 0,C 180,E1 23231.438,E2 23231.438} C_VEL
LIN {X 0,Y 599.961,Z 508.311,A -85,B 0,C 180,E1 23228.24,E2 23228.24} C_VEL
LIN {X 0,Y 599.965,Z 508.307,A -85,B 0,C 180,E1 23225.067,E2 23225.067} C_VEL
LIN {X 0,Y 599.96,Z 508.314,A -85,B 0,C 180,E1 23221.91,E2 23221.91} C_VEL
LIN {X 0,Y 599.968,Z 508.306,A -85,B 0,C 180,E1 23218.758,E2 23218.758} C_VEL
LIN {X 0,Y 599.956,Z 508.313,A -85,B 0,C 180,E1 23215.507,E2 23215.507} C_VEL
LIN {X 0,Y 599.958,Z 508.312,A -85,B 0,C 180,E1 23213.429,E2 23213.429} C_VEL
LIN {X 0,Y 598.952,Z 508.434,A -85,B 0,C 180,E1 23212.694,E2 23212.694} C_VEL
LIN {X 0,Y 592.557,Z 509.23,A -85,B 0,C 180,E1 23210.63,E2 23210.63} C_VEL
LIN {X 0,Y 592.022,Z 509.298,A -85,B 0,C 180,E1 23210.093,E2 23210.093} C_VEL
LIN {X 0,Y 592.012,Z 509.297,A -85,B 0,C 180,E1 23206.92,E2 23206.92} C_VEL
LIN {X 0,Y 592.023,Z 509.299,A -85,B 0,C 180,E1 23203.718,E2 23203.718} C_VEL
LIN {X 0,Y 592.011,Z 509.297,A -85,B 0,C 180,E1 23200.566,E2 23200.566} C_VEL
LIN {X 0,Y 592.024,Z 509.298,A -85,B 0,C 180,E1 23197.457,E2 23197.457} C_VEL
LIN {X 0,Y 592.011,Z 509.298,A -85,B 0,C 180,E1 23194.275,E2 23194.275} C_VEL
LIN {X 0,Y 592.027,Z 509.298,A -85,B 0,C 180,E1 23191.117,E2 23191.117} C_VEL
LIN {X 0,Y 592.011,Z 509.301,A -85,B 0,C 180,E1 23187.973,E2 23187.973} C_VEL
LIN {X 0,Y 592.029,Z 509.295,A -85,B 0,C 180,E1 23184.827,E2 23184.827} C_VEL
LIN {X 0,Y 592.009,Z 509.301,A -85,B 0,C 180,E1 23181.597,E2 23181.597} C_VEL
LIN {X 0,Y 592.027,Z 509.297,A -85,B 0,C 180,E1 23178.415,E2 23178.415} C_VEL
LIN {X 0,Y 592.007,Z 509.302,A -85,B 0,C 180,E1 23175.228,E2 23175.228} C_VEL
LIN {X 0,Y 592.029,Z 509.292,A -85,B 0,C 180,E1 23172.104,E2 23172.104} C_VEL
LIN {X 0,Y 592.004,Z 509.278,A -85,B 0,C 180,E1 23168.924,E2 23168.924} C_VEL
LIN {X 0,Y 592.082,Z 509.769,A -85,B 0,C 180,E1 23168.54,E2 23168.54} C_VEL
LIN {X 0,Y 594.409,Z 515.535,A -85,B 0,C 180,E1 23167.956,E2 23167.956} C_VEL
LIN {X 0,Y 594.037,Z 561.59,A -85,B 0,C 180,E1 23164.968,E2 23164.968} C_VEL
LIN {X 0,Y 593.961,Z 590.433,A -85,B 0,C 180,E1 23163.173,E2 23163.173} C_VEL
LIN {X 0,Y 594.409,Z 594.869,A -85,B 0,C 180,E1 23163.081,E2 23163.081} C_VEL
LIN {X 0,Y 593.958,Z 823.41,A -85,B 0,C 180,E1 23159.932,E2 23159.932} C_VEL
LIN {X 0,Y 593.81,Z 896.528,A -85,B 0,C 180,E1 23158.914,E2 23158.914} C_VEL
LIN {X 0,Y 593.689,Z 917.5,A -85,B 0,C 180,E1 23158.44,E2 23158.44} C_VEL
LIN {X 0,Y 593.518,Z 938.775,A -85,B 0,C 180,E1 23157.789,E2 23157.789} C_VEL
LIN {X 0,Y 593.38,Z 958.561,A -85,B 0,C 180,E1 23157.008,E2 23157.008} C_VEL
LIN {X 0,Y 593.182,Z 978.356,A -85,B 0,C 180,E1 23156.049,E2 23156.049} C_VEL
LIN {X 0,Y 593.003,Z 997.728,A -85,B 0,C 180,E1 23154.931,E2 23154.931} C_VEL
LIN {X 0,Y 592.807,Z 1016.17,A -85,B 0,C 180,E1 23153.667,E2 23153.667} C_VEL
LIN {X 0,Y 592.599,Z 1034.459,A -85,B 0,C 180,E1 23152.206,E2 23152.206} C_VEL
LIN {X 0,Y 592.419,Z 1051.479,A -85,B 0,C 180,E1 23150.628,E2 23150.628} C_VEL
LIN {X 0,Y 592.304,Z 1066.589,A -85,B 0,C 180,E1 23149.014,E2 23149.014} C_VEL
LIN {X 0,Y 592.178,Z 1081.268,A -85,B 0,C 180,E1 23147.186,E2 23147.186} C_VEL
LIN {X 0,Y 592.071,Z 1093.846,A -85,B 0,C 180,E1 23145.361,E2 23145.361} C_VEL
LIN {X 0,Y 592,Z 1104.996,A -85,B 0,C 180,E1 23143.478,E2 23143.478} C_VEL
LIN {X 0,Y 591.952,Z 1114.461,A -85,B 0,C 180,E1 23141.572,E2 23141.572} C_VEL
LIN {X 0,Y 591.918,Z 1122.801,A -85,B 0,C 180,E1 23139.529,E2 23139.529} C_VEL
LIN {X 0,Y 591.911,Z 1129.244,A -85,B 0,C 180,E1 23137.571,E2 23137.571} C_VEL
LIN {X 0,Y 591.912,Z 1134.214,A -85,B 0,C 180,E1 23135.525,E2 23135.525} C_VEL
LIN {X 0,Y 591.916,Z 1137.853,A -85,B 0,C 180,E1 23133.329,E2 23133.329} C_VEL
LIN {X 0,Y 591.905,Z 1139.683,A -85,B 0,C 180,E1 23131.258,E2 23131.258} C_VEL
LIN {X 0,Y 591.894,Z 1139.839,A -85,B 0,C 180,E1 23129.226,E2 23129.226} C_VEL
LIN {X 0,Y 591.892,Z 1138.448,A -85,B 0,C 180,E1 23127.095,E2 23127.095} C_VEL
LIN {X 0,Y 591.898,Z 1135.719,A -85,B 0,C 180,E1 23125.155,E2 23125.155} C_VEL
LIN {X 0,Y 591.917,Z 1131.269,A -85,B 0,C 180,E1 23123.112,E2 23123.112} C_VEL
LIN {X 0,Y 591.938,Z 1125.254,A -85,B 0,C 180,E1 23121.06,E2 23121.06} C_VEL
LIN {X 0,Y 591.953,Z 1117.751,A -85,B 0,C 180,E1 23119.095,E2 23119.095} C_VEL
LIN {X 0,Y 592.001,Z 1108.063,A -85,B 0,C 180,E1 23117.019,E2 23117.019} C_VEL
LIN {X 0,Y 592.065,Z 1097.519,A -85,B 0,C 180,E1 23115.126,E2 23115.126} C_VEL
LIN {X 0,Y 592.121,Z 1085.557,A -85,B 0,C 180,E1 23113.318,E2 23113.318} C_VEL
LIN {X 0,Y 592.244,Z 1071.59,A -85,B 0,C 180,E1 23111.495,E2 23111.495} C_VEL
LIN {X 0,Y 592.396,Z 1056.472,A -85,B 0,C 180,E1 23109.79,E2 23109.79} C_VEL
LIN {X 0,Y 592.574,Z 1039.376,A -85,B 0,C 180,E1 23108.129,E2 23108.129} C_VEL
LIN {X 0,Y 592.731,Z 1021.528,A -85,B 0,C 180,E1 23106.646,E2 23106.646} C_VEL
LIN {X 0,Y 592.939,Z 1002.312,A -85,B 0,C 180,E1 23105.279,E2 23105.279} C_VEL
LIN {X 0,Y 593.159,Z 983.056,A -85,B 0,C 180,E1 23104.114,E2 23104.114} C_VEL
LIN {X 0,Y 593.298,Z 964.109,A -85,B 0,C 180,E1 23103.15,E2 23103.15} C_VEL
LIN {X 0,Y 593.497,Z 943.402,A -85,B 0,C 180,E1 23102.291,E2 23102.291} C_VEL
LIN {X 0,Y 593.68,Z 922.436,A -85,B 0,C 180,E1 23101.6,E2 23101.6} C_VEL
LIN {X 0,Y 593.765,Z 901.803,A -85,B 0,C 180,E1 23101.103,E2 23101.103} C_VEL
LIN {X 0,Y 593.882,Z 874.315,A -85,B 0,C 180,E1 23100.668,E2 23100.668} C_VEL
LIN {X 0,Y 594.314,Z 645.666,A -85,B 0,C 180,E1 23097.538,E2 23097.538} C_VEL
LIN {X 0,Y 594.175,Z 593.252,A -85,B 0,C 180,E1 23096.792,E2 23096.792} C_VEL
LIN {X 0,Y 593.654,Z 589.931,A -85,B 0,C 180,E1 23096.656,E2 23096.656} C_VEL
LIN {X 0,Y 593.963,Z 550.726,A -85,B 0,C 180,E1 23093.662,E2 23093.662} C_VEL
LIN {X 0,Y 594.252,Z 515.4,A -85,B 0,C 180,E1 23090.865,E2 23090.865} C_VEL
LIN {X 0,Y 592.022,Z 509.502,A -85,B 0,C 180,E1 23090.17,E2 23090.17} C_VEL
LIN {X 0,Y 592,Z 509.299,A -85,B 0,C 180,E1 23086.973,E2 23086.973} C_VEL
LIN {X 0,Y 591.974,Z 509.302,A -85,B 0,C 180,E1 23084.097,E2 23084.097} C_VEL
LIN {X 0,Y 592.032,Z 509.299,A -85,B 0,C 180,E1 23080.941,E2 23080.941} C_VEL
LIN {X 0,Y 591.967,Z 509.303,A -85,B 0,C 180,E1 23077.928,E2 23077.928} C_VEL
LIN {X 0,Y 592.039,Z 509.293,A -85,B 0,C 180,E1 23074.808,E2 23074.808} C_VEL
LIN {X 0,Y 592.011,Z 509.611,A -85,B 0,C 180,E1 23073.553,E2 23073.553} C_VEL
LIN {X 0,Y 593.599,Z 514.945,A -85,B 0,C 180,E1 23073.013,E2 23073.013} C_VEL
LIN {X 0,Y 593.268,Z 551.939,A -85,B 0,C 180,E1 23070.148,E2 23070.148} C_VEL
LIN {X 0,Y 593.072,Z 592.25,A -85,B 0,C 180,E1 23067.107,E2 23067.107} C_VEL
LIN {X 0,Y 592.816,Z 635.765,A -85,B 0,C 180,E1 23063.914,E2 23063.914} C_VEL
LIN {X 0,Y 592.576,Z 679.87,A -85,B 0,C 180,E1 23060.753,E2 23060.753} C_VEL
LIN {X 0,Y 592.511,Z 705.598,A -85,B 0,C 180,E1 23058.967,E2 23058.967} C_VEL
LIN {X 0,Y 592.579,Z 820.678,A -85,B 0,C 180,E1 23057.523,E2 23057.523} C_VEL
LIN {X 0,Y 592.563,Z 876.343,A -85,B 0,C 180,E1 23056.802,E2 23056.802} C_VEL
LIN {X 0,Y 592.508,Z 893.896,A -85,B 0,C 180,E1 23056.388,E2 23056.388} C_VEL
LIN {X 0,Y 592.418,Z 910.814,A -85,B 0,C 180,E1 23055.804,E2 23055.804} C_VEL
LIN {X 0,Y 592.337,Z 926.741,A -85,B 0,C 180,E1 23055.067,E2 23055.067} C_VEL
LIN {X 0,Y 592.255,Z 941.921,A -85,B 0,C 180,E1 23054.17,E2 23054.17} C_VEL
LIN {X 0,Y 592.162,Z 956.701,A -85,B 0,C 180,E1 23053.077,E2 23053.077} C_VEL
LIN {X 0,Y 592.09,Z 970.313,A -85,B 0,C 180,E1 23051.84,E2 23051.84} C_VEL
LIN {X 0,Y 592.018,Z 982.182,A -85,B 0,C 180,E1 23050.51,E2 23050.51} C_VEL
LIN {X 0,Y 591.972,Z 992.832,A -85,B 0,C 180,E1 23049.038,E2 23049.038} C_VEL
LIN {X 0,Y 591.945,Z 1001.854,A -85,B 0,C 180,E1 23047.473,E2 23047.473} C_VEL
LIN {X 0,Y 591.923,Z 1008.814,A -85,B 0,C 180,E1 23045.914,E2 23045.914} C_VEL
LIN {X 0,Y 591.916,Z 1014.212,A -85,B 0,C 180,E1 23044.263,E2 23044.263} C_VEL
LIN {X 0,Y 591.913,Z 1017.792,A -85,B 0,C 180,E1 23042.614,E2 23042.614} C_VEL
LIN {X 0,Y 591.913,Z 1019.722,A -85,B 0,C 180,E1 23040.871,E2 23040.871} C_VEL
LIN {X 0,Y 591.916,Z 1019.82,A -85,B 0,C 180,E1 23039.226,E2 23039.226} C_VEL
LIN {X 0,Y 591.912,Z 1018.252,A -85,B 0,C 180,E1 23037.58,E2 23037.58} C_VEL
LIN {X 0,Y 591.913,Z 1014.953,A -85,B 0,C 180,E1 23035.932,E2 23035.932} C_VEL
LIN {X 0,Y 591.924,Z 1009.842,A -85,B 0,C 180,E1 23034.281,E2 23034.281} C_VEL
LIN {X 0,Y 591.938,Z 1003.255,A -85,B 0,C 180,E1 23032.722,E2 23032.722} C_VEL
LIN {X 0,Y 591.966,Z 994.632,A -85,B 0,C 180,E1 23031.151,E2 23031.151} C_VEL
LIN {X 0,Y 592.012,Z 984.444,A -85,B 0,C 180,E1 23029.687,E2 23029.687} C_VEL
LIN {X 0,Y 592.07,Z 972.605,A -85,B 0,C 180,E1 23028.308,E2 23028.308} C_VEL
LIN {X 0,Y 592.143,Z 960.144,A -85,B 0,C 180,E1 23027.122,E2 23027.122} C_VEL
LIN {X 0,Y 592.233,Z 946.153,A -85,B 0,C 180,E1 23026.03,E2 23026.03} C_VEL
LIN {X 0,Y 592.301,Z 930.198,A -85,B 0,C 180,E1 23025.032,E2 23025.032} C_VEL
LIN {X 0,Y 592.388,Z 914.971,A -85,B 0,C 180,E1 23024.283,E2 23024.283} C_VEL
LIN {X 0,Y 592.492,Z 898.424,A -85,B 0,C 180,E1 23023.657,E2 23023.657} C_VEL
LIN {X 0,Y 592.56,Z 881.002,A -85,B 0,C 180,E1 23023.198,E2 23023.198} C_VEL
LIN {X 0,Y 592.571,Z 859.387,A -85,B 0,C 180,E1 23022.869,E2 23022.869} C_VEL
LIN {X 0,Y 592.563,Z 705.925,A -85,B 0,C 180,E1 23020.946,E2 23020.946} C_VEL
LIN {X 0,Y 592.44,Z 703.691,A -85,B 0,C 180,E1 23020.837,E2 23020.837} C_VEL
LIN {X 0,Y 592.698,Z 660.283,A -85,B 0,C 180,E1 23017.762,E2 23017.762} C_VEL
LIN {X 0,Y 592.925,Z 615.679,A -85,B 0,C 180,E1 23014.532,E2 23014.532} C_VEL
LIN {X 0,Y 593.122,Z 575.67,A -85,B 0,C 180,E1 23011.561,E2 23011.561} C_VEL
LIN {X 0,Y 593.485,Z 530.508,A -85,B 0,C 180,E1 23008.115,E2 23008.115} C_VEL
LIN {X 0,Y 593.456,Z 513.835,A -85,B 0,C 180,E1 23006.801,E2 23006.801} C_VEL
LIN {X 0,Y 592.001,Z 509.54,A -85,B 0,C 180,E1 23006.331,E2 23006.331} C_VEL
LIN {X 0,Y 592.026,Z 509.307,A -85,B 0,C 180,E1 23003.505,E2 23003.505} C_VEL
LIN {X 0,Y 592.006,Z 509.294,A -85,B 0,C 180,E1 23000.327,E2 23000.327} C_VEL
LIN {X 0,Y 592.023,Z 509.301,A -85,B 0,C 180,E1 22997.24,E2 22997.24} C_VEL
LIN {X 0,Y 592.029,Z 509.302,A -85,B 0,C 180,E1 22994.092,E2 22994.092} C_VEL
LIN {X 0,Y 592.019,Z 509.456,A -85,B 0,C 180,E1 22991.181,E2 22991.181} C_VEL
LIN {X 0,Y 593.102,Z 512.467,A -85,B 0,C 180,E1 22990.806,E2 22990.806} C_VEL
LIN {X 0,Y 594.564,Z 516.017,A -85,B 0,C 180,E1 22990.412,E2 22990.412} C_VEL
LIN {X 0,Y 594.385,Z 543.506,A -85,B 0,C 180,E1 22988.369,E2 22988.369} C_VEL
LIN {X 0,Y 595.205,Z 548.226,A -85,B 0,C 180,E1 22988.227,E2 22988.227} C_VEL
LIN {X 0,Y 594.729,Z 756.058,A -85,B 0,C 180,E1 22985.196,E2 22985.196} C_VEL
LIN {X 0,Y 594.413,Z 891.439,A -85,B 0,C 180,E1 22983.25,E2 22983.25} C_VEL
LIN {X 0,Y 594.253,Z 915.113,A -85,B 0,C 180,E1 22982.726,E2 22982.726} C_VEL
LIN {X 0,Y 594.111,Z 935.243,A -85,B 0,C 180,E1 22982.121,E2 22982.121} C_VEL
LIN {X 0,Y 593.861,Z 958.397,A -85,B 0,C 180,E1 22981.236,E2 22981.236} C_VEL
LIN {X 0,Y 593.682,Z 978.538,A -85,B 0,C 180,E1 22980.292,E2 22980.292} C_VEL
LIN {X 0,Y 593.399,Z 1000.14,A -85,B 0,C 180,E1 22979.086,E2 22979.086} C_VEL
LIN {X 0,Y 593.193,Z 1020.455,A -85,B 0,C 180,E1 22977.76,E2 22977.76} C_VEL
LIN {X 0,Y 592.93,Z 1039.255,A -85,B 0,C 180,E1 22976.327,E2 22976.327} C_VEL
LIN {X 0,Y 592.699,Z 1058.325,A -85,B 0,C 180,E1 22974.671,E2 22974.671} C_VEL
LIN {X 0,Y 592.524,Z 1075.351,A -85,B 0,C 180,E1 22972.975,E2 22972.975} C_VEL
LIN {X 0,Y 592.349,Z 1091.136,A -85,B 0,C 180,E1 22971.175,E2 22971.175} C_VEL
LIN {X 0,Y 592.236,Z 1105.582,A -85,B 0,C 180,E1 22969.311,E2 22969.311} C_VEL
LIN {X 0,Y 592.125,Z 1118.448,A -85,B 0,C 180,E1 22967.391,E2 22967.391} C_VEL
LIN {X 0,Y 592.031,Z 1130.75,A -85,B 0,C 180,E1 22965.276,E2 22965.276} C_VEL
LIN {X 0,Y 591.962,Z 1140.186,A -85,B 0,C 180,E1 22963.372,E2 22963.372} C_VEL
LIN {X 0,Y 591.935,Z 1149.268,A -85,B 0,C 180,E1 22961.201,E2 22961.201} C_VEL
LIN {X 0,Y 591.918,Z 1155.953,A -85,B 0,C 180,E1 22959.234,E2 22959.234} C_VEL
LIN {X 0,Y 591.888,Z 1161.807,A -85,B 0,C 180,E1 22957.084,E2 22957.084} C_VEL
LIN {X 0,Y 591.907,Z 1165.957,A -85,B 0,C 180,E1 22954.942,E2 22954.942} C_VEL
LIN {X 0,Y 591.896,Z 1168.718,A -85,B 0,C 180,E1 22952.808,E2 22952.808} C_VEL
LIN {X 0,Y 591.882,Z 1169.85,A -85,B 0,C 180,E1 22950.678,E2 22950.678} C_VEL
LIN {X 0,Y 591.91,Z 1169.657,A -85,B 0,C 180,E1 22948.548,E2 22948.548} C_VEL
LIN {X 0,Y 591.894,Z 1167.841,A -85,B 0,C 180,E1 22946.417,E2 22946.417} C_VEL
LIN {X 0,Y 591.891,Z 1164.627,A -85,B 0,C 180,E1 22944.249,E2 22944.249} C_VEL
LIN {X 0,Y 591.918,Z 1159.57,A -85,B 0,C 180,E1 22942.038,E2 22942.038} C_VEL
LIN {X 0,Y 591.928,Z 1153.182,A -85,B 0,C 180,E1 22939.882,E2 22939.882} C_VEL
LIN {X 0,Y 591.94,Z 1145.332,A -85,B 0,C 180,E1 22937.811,E2 22937.811} C_VEL
LIN {X 0,Y 592.008,Z 1135.951,A -85,B 0,C 180,E1 22935.725,E2 22935.725} C_VEL
LIN {X 0,Y 592.067,Z 1125.135,A -85,B 0,C 180,E1 22933.72,E2 22933.72} C_VEL
LIN {X 0,Y 592.164,Z 1112.578,A -85,B 0,C 180,E1 22931.696,E2 22931.696} C_VEL
LIN {X 0,Y 592.26,Z 1099.092,A -85,B 0,C 180,E1 22929.824,E2 22929.824} C_VEL
LIN {X 0,Y 592.433,Z 1082.73,A -85,B 0,C 180,E1 22927.839,E2 22927.839} C_VEL
LIN {X 0,Y 592.639,Z 1066.53,A -85,B 0,C 180,E1 22926.114,E2 22926.114} C_VEL
LIN {X 0,Y 592.806,Z 1048.752,A -85,B 0,C 180,E1 22924.469,E2 22924.469} C_VEL
LIN {X 0,Y 593.065,Z 1029.301,A -85,B 0,C 180,E1 22922.893,E2 22922.893} C_VEL
LIN {X 0,Y 593.282,Z 1010.554,A -85,B 0,C 180,E1 22921.569,E2 22921.569} C_VEL
LIN {X 0,Y 593.538,Z 989.806,A -85,B 0,C 180,E1 22920.313,E2 22920.313} C_VEL
LIN {X 0,Y 593.755,Z 969.581,A -85,B 0,C 180,E1 22919.264,E2 22919.264} C_VEL
LIN {X 0,Y 593.989,Z 947.393,A -85,B 0,C 180,E1 22918.319,E2 22918.319} C_VEL
LIN {X 0,Y 594.177,Z 925.969,A -85,B 0,C 180,E1 22917.577,E2 22917.577} C_VEL
LIN {X 0,Y 594.335,Z 903.589,A -85,B 0,C 180,E1 22916.996,E2 22916.996} C_VEL
LIN {X 0,Y 594.435,Z 883.308,A -85,B 0,C 180,E1 22916.615,E2 22916.615} C_VEL
LIN {X 0,Y 594.922,Z 666.768,A -85,B 0,C 180,E1 22913.515,E2 22913.515} C_VEL
LIN {X 0,Y 595.059,Z 544.959,A -85,B 0,C 180,E1 22911.712,E2 22911.712} C_VEL
LIN {X 0,Y 594.559,Z 541.755,A -85,B 0,C 180,E1 22911.597,E2 22911.597} C_VEL
LIN {X 0,Y 594.722,Z 515.838,A -85,B 0,C 180,E1 22909.985,E2 22909.985} C_VEL
LIN {X 0,Y 592.074,Z 509.68,A -85,B 0,C 180,E1 22909.342,E2 22909.342} C_VEL
LIN {X 0,Y 592.031,Z 509.262,A -85,B 0,C 180,E1 22908.674,E2 22908.674} C_VEL
LIN {X 0,Y 592.025,Z 509.297,A -85,B 0,C 180,E1 22905.317,E2 22905.317} C_VEL
LIN {X 0,Y 592.029,Z 509.302,A -85,B 0,C 180,E1 22902.104,E2 22902.104} C_VEL
LIN {X 0,Y 592.017,Z 509.298,A -85,B 0,C 180,E1 22898.798,E2 22898.798} C_VEL
LIN {X 0,Y 592.023,Z 509.302,A -85,B 0,C 180,E1 22895.638,E2 22895.638} C_VEL
LIN {X 0,Y 592.019,Z 509.294,A -85,B 0,C 180,E1 22892.484,E2 22892.484} C_VEL
LIN {X 0,Y 592.022,Z 509.301,A -85,B 0,C 180,E1 22889.326,E2 22889.326} C_VEL
LIN {X 0,Y 592.02,Z 509.294,A -85,B 0,C 180,E1 22886.155,E2 22886.155} C_VEL
LIN {X 0,Y 592.02,Z 509.298,A -85,B 0,C 180,E1 22882.962,E2 22882.962} C_VEL
LIN {X 0,Y 592.019,Z 509.296,A -85,B 0,C 180,E1 22879.741,E2 22879.741} C_VEL
LIN {X 0,Y 592.019,Z 509.297,A -85,B 0,C 180,E1 22876.584,E2 22876.584} C_VEL
LIN {X 0,Y 592.02,Z 509.295,A -85,B 0,C 180,E1 22873.392,E2 22873.392} C_VEL
LIN {X 0,Y 592.017,Z 509.297,A -85,B 0,C 180,E1 22870.214,E2 22870.214} C_VEL
LIN {X 0,Y 592.022,Z 509.294,A -85,B 0,C 180,E1 22867.082,E2 22867.082} C_VEL
LIN {X 0,Y 592.016,Z 509.299,A -85,B 0,C 180,E1 22863.873,E2 22863.873} C_VEL
LIN {X 0,Y 592.021,Z 509.298,A -85,B 0,C 180,E1 22860.677,E2 22860.677} C_VEL
LIN {X 0,Y 592.014,Z 509.3,A -85,B 0,C 180,E1 22857.483,E2 22857.483} C_VEL
LIN {X 0,Y 592.021,Z 509.299,A -85,B 0,C 180,E1 22854.281,E2 22854.281} C_VEL
LIN {X 0,Y 592.013,Z 509.3,A -85,B 0,C 180,E1 22851.122,E2 22851.122} C_VEL
LIN {X 0,Y 592.022,Z 509.298,A -85,B 0,C 180,E1 22850.093,E2 22850.093} C_VEL
LIN {X 0,Y 591.024,Z 509.428,A -85,B 0,C 180,E1 22849.347,E2 22849.347} C_VEL
LIN {X 0,Y 584.598,Z 510.224,A -85,B 0,C 180,E1 22847.255,E2 22847.255} C_VEL
LIN {X 0,Y 584.074,Z 510.283,A -85,B 0,C 180,E1 22846.711,E2 22846.711} C_VEL
LIN {X 0,Y 584.088,Z 510.291,A -85,B 0,C 180,E1 22843.462,E2 22843.462} C_VEL
LIN {X 0,Y 584.075,Z 510.282,A -85,B 0,C 180,E1 22840.291,E2 22840.291} C_VEL
LIN {X 0,Y 584.091,Z 510.292,A -85,B 0,C 180,E1 22837.027,E2 22837.027} C_VEL
LIN {X 0,Y 584.083,Z 510.281,A -85,B 0,C 180,E1 22833.768,E2 22833.768} C_VEL
LIN {X 0,Y 584.087,Z 510.288,A -85,B 0,C 180,E1 22830.349,E2 22830.349} C_VEL
LIN {X 0,Y 584.093,Z 510.285,A -85,B 0,C 180,E1 22827.013,E2 22827.013} C_VEL
LIN {X 0,Y 584.072,Z 510.289,A -85,B 0,C 180,E1 22823.736,E2 22823.736} C_VEL
LIN {X 0,Y 584.089,Z 510.286,A -85,B 0,C 180,E1 22820.537,E2 22820.537} C_VEL
LIN {X 0,Y 584.069,Z 510.289,A -85,B 0,C 180,E1 22817.32,E2 22817.32} C_VEL
LIN {X 0,Y 584.09,Z 510.289,A -85,B 0,C 180,E1 22814.164,E2 22814.164} C_VEL
LIN {X 0,Y 584.068,Z 510.295,A -85,B 0,C 180,E1 22810.969,E2 22810.969} C_VEL
LIN {X 0,Y 584.106,Z 510.472,A -85,B 0,C 180,E1 22809.155,E2 22809.155} C_VEL
LIN {X 0,Y 585.144,Z 513.407,A -85,B 0,C 180,E1 22808.814,E2 22808.814} C_VEL
LIN {X 0,Y 587.674,Z 519.468,A -85,B 0,C 180,E1 22808.204,E2 22808.204} C_VEL
LIN {X 0,Y 587.117,Z 565.755,A -85,B 0,C 180,E1 22805.171,E2 22805.171} C_VEL
LIN {X 0,Y 586.976,Z 590.47,A -85,B 0,C 180,E1 22803.62,E2 22803.62} C_VEL
LIN {X 0,Y 587.703,Z 595.854,A -85,B 0,C 180,E1 22803.494,E2 22803.494} C_VEL
LIN {X 0,Y 587.023,Z 824.238,A -85,B 0,C 180,E1 22800.311,E2 22800.311} C_VEL
LIN {X 0,Y 586.802,Z 896.676,A -85,B 0,C 180,E1 22799.291,E2 22799.291} C_VEL
LIN {X 0,Y 586.614,Z 917.813,A -85,B 0,C 180,E1 22798.807,E2 22798.807} C_VEL
LIN {X 0,Y 586.361,Z 939.383,A -85,B 0,C 180,E1 22798.136,E2 22798.136} C_VEL
LIN {X 0,Y 586.141,Z 959.852,A -85,B 0,C 180,E1 22797.314,E2 22797.314} C_VEL
LIN {X 0,Y 585.837,Z 979.417,A -85,B 0,C 180,E1 22796.343,E2 22796.343} C_VEL
LIN {X 0,Y 585.54,Z 999.358,A -85,B 0,C 180,E1 22795.163,E2 22795.163} C_VEL
LIN {X 0,Y 585.259,Z 1018.361,A -85,B 0,C 180,E1 22793.831,E2 22793.831} C_VEL
LIN {X 0,Y 584.949,Z 1036.08,A -85,B 0,C 180,E1 22792.371,E2 22792.371} C_VEL
LIN {X 0,Y 584.673,Z 1053.244,A -85,B 0,C 180,E1 22790.732,E2 22790.732} C_VEL
LIN {X 0,Y 584.461,Z 1069.147,A -85,B 0,C 180,E1 22788.968,E2 22788.968} C_VEL
LIN {X 0,Y 584.309,Z 1082.806,A -85,B 0,C 180,E1 22787.22,E2 22787.22} C_VEL
LIN {X 0,Y 584.157,Z 1095.685,A -85,B 0,C 180,E1 22785.283,E2 22785.283} C_VEL
LIN {X 0,Y 584.048,Z 1107.078,A -85,B 0,C 180,E1 22783.262,E2 22783.262} C_VEL
LIN {X 0,Y 583.983,Z 1116.567,A -85,B 0,C 180,E1 22781.255,E2 22781.255} C_VEL
LIN {X 0,Y 583.933,Z 1124.223,A -85,B 0,C 180,E1 22779.262,E2 22779.262} C_VEL
LIN {X 0,Y 583.903,Z 1130.529,A -85,B 0,C 180,E1 22777.181,E2 22777.181} C_VEL
LIN {X 0,Y 583.897,Z 1135.039,A -85,B 0,C 180,E1 22775.207,E2 22775.207} C_VEL
LIN {X 0,Y 583.905,Z 1138.12,A -85,B 0,C 180,E1 22773.141,E2 22773.141} C_VEL
LIN {X 0,Y 583.909,Z 1139.773,A -85,B 0,C 180,E1 22770.981,E2 22770.981} C_VEL
LIN {X 0,Y 583.911,Z 1139.772,A -85,B 0,C 180,E1 22768.921,E2 22768.921} C_VEL
LIN {X 0,Y 583.905,Z 1138.111,A -85,B 0,C 180,E1 22766.761,E2 22766.761} C_VEL
LIN {X 0,Y 583.899,Z 1135.02,A -85,B 0,C 180,E1 22764.694,E2 22764.694} C_VEL
LIN {X 0,Y 583.904,Z 1130.506,A -85,B 0,C 180,E1 22762.72,E2 22762.72} C_VEL
LIN {X 0,Y 583.931,Z 1123.834,A -85,B 0,C 180,E1 22760.539,E2 22760.539} C_VEL
LIN {X 0,Y 583.982,Z 1116.118,A -85,B 0,C 180,E1 22758.544,E2 22758.544} C_VEL
LIN {X 0,Y 584.046,Z 1106.503,A -85,B 0,C 180,E1 22756.536,E2 22756.536} C_VEL
LIN {X 0,Y 584.154,Z 1094.917,A -85,B 0,C 180,E1 22754.505,E2 22754.505} C_VEL
LIN {X 0,Y 584.306,Z 1082.714,A -85,B 0,C 180,E1 22752.678,E2 22752.678} C_VEL
LIN {X 0,Y 584.482,Z 1068.183,A -85,B 0,C 180,E1 22750.825,E2 22750.825} C_VEL
LIN {X 0,Y 584.683,Z 1052.597,A -85,B 0,C 180,E1 22749.111,E2 22749.111} C_VEL
LIN {X 0,Y 584.962,Z 1034.89,A -85,B 0,C 180,E1 22747.435,E2 22747.435} C_VEL
LIN {X 0,Y 585.266,Z 1017.404,A -85,B 0,C 180,E1 22746.009,E2 22746.009} C_VEL
LIN {X 0,Y 585.547,Z 999.086,A -85,B 0,C 180,E1 22744.729,E2 22744.729} C_VEL
LIN {X 0,Y 585.839,Z 979.069,A -85,B 0,C 180,E1 22743.548,E2 22743.548} C_VEL
LIN {X 0,Y 586.146,Z 959.391,A -85,B 0,C 180,E1 22742.576,E2 22742.576} C_VEL
LIN {X 0,Y 586.374,Z 938.974,A -85,B 0,C 180,E1 22741.759,E2 22741.759} C_VEL
LIN {X 0,Y 586.616,Z 917.221,A -85,B 0,C 180,E1 22741.087,E2 22741.087} C_VEL
LIN {X 0,Y 586.805,Z 896.082,A -85,B 0,C 180,E1 22740.61,E2 22740.61} C_VEL
LIN {X 0,Y 587.108,Z 799.135,A -85,B 0,C 180,E1 22739.254,E2 22739.254} C_VEL
LIN {X 0,Y 587.623,Z 595.59,A -85,B 0,C 180,E1 22736.407,E2 22736.407} C_VEL
LIN {X 0,Y 586.603,Z 590.541,A -85,B 0,C 180,E1 22736.243,E2 22736.243} C_VEL
LIN {X 0,Y 587.068,Z 550.716,A -85,B 0,C 180,E1 22733.165,E2 22733.165} C_VEL
LIN {X 0,Y 587.376,Z 518.908,A -85,B 0,C 180,E1 22730.608,E2 22730.608} C_VEL
LIN {X 0,Y 584.136,Z 510.535,A -85,B 0,C 180,E1 22729.615,E2 22729.615} C_VEL
LIN {X 0,Y 584.035,Z 510.289,A -85,B 0,C 180,E1 22726.51,E2 22726.51} C_VEL
LIN {X 0,Y 584.091,Z 510.282,A -85,B 0,C 180,E1 22723.463,E2 22723.463} C_VEL
LIN {X 0,Y 584.036,Z 510.294,A -85,B 0,C 180,E1 22720.326,E2 22720.326} C_VEL
LIN {X 0,Y 584.056,Z 510.291,A -85,B 0,C 180,E1 22717.407,E2 22717.407} C_VEL
LIN {X 0,Y 584.041,Z 510.287,A -85,B 0,C 180,E1 22714.162,E2 22714.162} C_VEL
LIN {X 0,Y 584.105,Z 510.795,A -85,B 0,C 180,E1 22713.854,E2 22713.854} C_VEL
LIN {X 0,Y 586.319,Z 517.226,A -85,B 0,C 180,E1 22713.248,E2 22713.248} C_VEL
LIN {X 0,Y 586.08,Z 548.242,A -85,B 0,C 180,E1 22710.847,E2 22710.847} C_VEL
LIN {X 0,Y 585.697,Z 586.837,A -85,B 0,C 180,E1 22707.889,E2 22707.889} C_VEL
LIN {X 0,Y 585.335,Z 630.004,A -85,B 0,C 180,E1 22704.666,E2 22704.666} C_VEL
LIN {X 0,Y 584.974,Z 672.183,A -85,B 0,C 180,E1 22701.592,E2 22701.592} C_VEL
LIN {X 0,Y 584.797,Z 705.504,A -85,B 0,C 180,E1 22699.229,E2 22699.229} C_VEL
LIN {X 0,Y 585.148,Z 712.63,A -85,B 0,C 180,E1 22699.123,E2 22699.123} C_VEL
LIN {X 0,Y 584.903,Z 875.904,A -85,B 0,C 180,E1 22697.038,E2 22697.038} C_VEL
LIN {X 0,Y 584.815,Z 893.594,A -85,B 0,C 180,E1 22696.619,E2 22696.619} C_VEL
LIN {X 0,Y 584.687,Z 911.016,A -85,B 0,C 180,E1 22696.011,E2 22696.011} C_VEL
LIN {X 0,Y 584.553,Z 927.592,A -85,B 0,C 180,E1 22695.227,E2 22695.227} C_VEL
LIN {X 0,Y 584.421,Z 942.99,A -85,B 0,C 180,E1 22694.29,E2 22694.29} C_VEL
LIN {X 0,Y 584.285,Z 957.919,A -85,B 0,C 180,E1 22693.156,E2 22693.156} C_VEL
LIN {X 0,Y 584.175,Z 970.805,A -85,B 0,C 180,E1 22691.953,E2 22691.953} C_VEL
LIN {X 0,Y 584.078,Z 982.187,A -85,B 0,C 180,E1 22690.654,E2 22690.654} C_VEL
LIN {X 0,Y 584.002,Z 992.839,A -85,B 0,C 180,E1 22689.162,E2 22689.162} C_VEL
LIN {X 0,Y 583.96,Z 1001.857,A -85,B 0,C 180,E1 22687.576,E2 22687.576} C_VEL
LIN {X 0,Y 583.932,Z 1008.814,A -85,B 0,C 180,E1 22685.996,E2 22685.996} C_VEL
LIN {X 0,Y 583.918,Z 1014.215,A -85,B 0,C 180,E1 22684.321,E2 22684.321} C_VEL
LIN {X 0,Y 583.914,Z 1017.796,A -85,B 0,C 180,E1 22682.65,E2 22682.65} C_VEL
LIN {X 0,Y 583.913,Z 1019.724,A -85,B 0,C 180,E1 22680.883,E2 22680.883} C_VEL
LIN {X 0,Y 583.916,Z 1019.813,A -85,B 0,C 180,E1 22679.215,E2 22679.215} C_VEL
LIN {X 0,Y 583.913,Z 1018.254,A -85,B 0,C 180,E1 22677.547,E2 22677.547} C_VEL
LIN {X 0,Y 583.914,Z 1014.954,A -85,B 0,C 180,E1 22675.876,E2 22675.876} C_VEL
LIN {X 0,Y 583.927,Z 1009.771,A -85,B 0,C 180,E1 22674.184,E2 22674.184} C_VEL
LIN {X 0,Y 583.952,Z 1003.254,A -85,B 0,C 180,E1 22672.622,E2 22672.622} C_VEL
LIN {X 0,Y 583.996,Z 994.671,A -85,B 0,C 180,E1 22671.037,E2 22671.037} C_VEL
LIN {X 0,Y 584.058,Z 985.198,A -85,B 0,C 180,E1 22669.645,E2 22669.645} C_VEL
LIN {X 0,Y 584.146,Z 973.529,A -85,B 0,C 180,E1 22668.248,E2 22668.248} C_VEL
LIN {X 0,Y 584.259,Z 960.767,A -85,B 0,C 180,E1 22667.001,E2 22667.001} C_VEL
LIN {X 0,Y 584.393,Z 946.861,A -85,B 0,C 180,E1 22665.889,E2 22665.889} C_VEL
LIN {X 0,Y 584.508,Z 931.08,A -85,B 0,C 180,E1 22664.879,E2 22664.879} C_VEL
LIN {X 0,Y 584.637,Z 916.069,A -85,B 0,C 180,E1 22664.12,E2 22664.12} C_VEL
LIN {X 0,Y 584.776,Z 899.894,A -85,B 0,C 180,E1 22663.486,E2 22663.486} C_VEL
LIN {X 0,Y 584.874,Z 882.698,A -85,B 0,C 180,E1 22663.01,E2 22663.01} C_VEL
LIN {X 0,Y 584.923,Z 864.213,A -85,B 0,C 180,E1 22662.699,E2 22662.699} C_VEL
LIN {X 0,Y 584.98,Z 706.842,A -85,B 0,C 180,E1 22660.708,E2 22660.708} C_VEL
LIN {X 0,Y 584.744,Z 704.422,A -85,B 0,C 180,E1 22660.627,E2 22660.627} C_VEL
LIN {X 0,Y 585.1,Z 661.496,A -85,B 0,C 180,E1 22657.547,E2 22657.547} C_VEL
LIN {X 0,Y 585.45,Z 617.124,A -85,B 0,C 180,E1 22654.292,E2 22654.292} C_VEL
LIN {X 0,Y 585.773,Z 577.117,A -85,B 0,C 180,E1 22651.283,E2 22651.283} C_VEL
LIN {X 0,Y 586.295,Z 532.012,A -85,B 0,C 180,E1 22647.797,E2 22647.797} C_VEL
LIN {X 0,Y 586.179,Z 516.878,A -85,B 0,C 180,E1 22646.66,E2 22646.66} C_VEL
LIN {X 0,Y 584.079,Z 510.633,A -85,B 0,C 180,E1 22646.167,E2 22646.167} C_VEL
LIN {X 0,Y 584.057,Z 510.299,A -85,B 0,C 180,E1 22645.722,E2 22645.722} C_VEL
LIN {X 0,Y 584.06,Z 510.29,A -85,B 0,C 180,E1 22642.431,E2 22642.431} C_VEL
LIN {X 0,Y 584.092,Z 510.284,A -85,B 0,C 180,E1 22639.293,E2 22639.293} C_VEL
LIN {X 0,Y 584.082,Z 510.286,A -85,B 0,C 180,E1 22636.109,E2 22636.109} C_VEL
LIN {X 0,Y 584.065,Z 510.283,A -85,B 0,C 180,E1 22632.948,E2 22632.948} C_VEL
LIN {X 0,Y 584.121,Z 510.455,A -85,B 0,C 180,E1 22631.782,E2 22631.782} C_VEL
LIN {X 0,Y 585.228,Z 513.538,A -85,B 0,C 180,E1 22631.391,E2 22631.391} C_VEL
LIN {X 0,Y 587.901,Z 519.882,A -85,B 0,C 180,E1 22630.666,E2 22630.666} C_VEL
LIN {X 0,Y 587.659,Z 543.54,A -85,B 0,C 180,E1 22628.89,E2 22628.89} C_VEL
LIN {X 0,Y 588.907,Z 549.986,A -85,B 0,C 180,E1 22628.685,E2 22628.685} C_VEL
LIN {X 0,Y 588.181,Z 757.357,A -85,B 0,C 180,E1 22625.628,E2 22625.628} C_VEL
LIN {X 0,Y 587.711,Z 891.546,A -85,B 0,C 180,E1 22623.677,E2 22623.677} C_VEL
LIN {X 0,Y 587.467,Z 915.284,A -85,B 0,C 180,E1 22623.147,E2 22623.147} C_VEL
LIN {X 0,Y 587.252,Z 936,A -85,B 0,C 180,E1 22622.517,E2 22622.517} C_VEL
LIN {X 0,Y 586.875,Z 959.122,A -85,B 0,C 180,E1 22621.618,E2 22621.618} C_VEL
LIN {X 0,Y 586.588,Z 980.559,A -85,B 0,C 180,E1 22620.595,E2 22620.595} C_VEL
LIN {X 0,Y 586.172,Z 1001.033,A -85,B 0,C 180,E1 22619.423,E2 22619.423} C_VEL
LIN {X 0,Y 585.846,Z 1021.34,A -85,B 0,C 180,E1 22618.072,E2 22618.072} C_VEL
LIN {X 0,Y 585.457,Z 1040.581,A -85,B 0,C 180,E1 22616.58,E2 22616.58} C_VEL
LIN {X 0,Y 585.096,Z 1059.989,A -85,B 0,C 180,E1 22614.851,E2 22614.851} C_VEL
LIN {X 0,Y 584.834,Z 1077.115,A -85,B 0,C 180,E1 22613.106,E2 22613.106} C_VEL
LIN {X 0,Y 584.568,Z 1093.141,A -85,B 0,C 180,E1 22611.224,E2 22611.224} C_VEL
LIN {X 0,Y 584.352,Z 1108.33,A -85,B 0,C 180,E1 22609.179,E2 22609.179} C_VEL
LIN {X 0,Y 584.216,Z 1121.643,A -85,B 0,C 180,E1 22607.12,E2 22607.12} C_VEL
LIN {X 0,Y 584.091,Z 1132.835,A -85,B 0,C 180,E1 22605.082,E2 22605.082} C_VEL
LIN {X 0,Y 584.009,Z 1142.878,A -85,B 0,C 180,E1 22602.961,E2 22602.961} C_VEL
LIN {X 0,Y 583.953,Z 1151.05,A -85,B 0,C 180,E1 22600.856,E2 22600.856} C_VEL
LIN {X 0,Y 583.936,Z 1158.039,A -85,B 0,C 180,E1 22598.666,E2 22598.666} C_VEL
LIN {X 0,Y 583.92,Z 1163.253,A -85,B 0,C 180,E1 22596.489,E2 22596.489} C_VEL
LIN {X 0,Y 583.916,Z 1167.163,A -85,B 0,C 180,E1 22594.223,E2 22594.223} C_VEL
LIN {X 0,Y 583.913,Z 1169.256,A -85,B 0,C 180,E1 22592.061,E2 22592.061} C_VEL
LIN {X 0,Y 583.9,Z 1169.962,A -85,B 0,C 180,E1 22589.804,E2 22589.804} C_VEL
LIN {X 0,Y 583.916,Z 1169.122,A -85,B 0,C 180,E1 22587.743,E2 22587.743} C_VEL
LIN {X 0,Y 583.904,Z 1166.753,A -85,B 0,C 180,E1 22585.482,E2 22585.482} C_VEL
LIN {X 0,Y 583.913,Z 1163.047,A -85,B 0,C 180,E1 22583.412,E2 22583.412} C_VEL
LIN {X 0,Y 583.936,Z 1157.775,A -85,B 0,C 180,E1 22581.234,E2 22581.234} C_VEL
LIN {X 0,Y 583.951,Z 1150.693,A -85,B 0,C 180,E1 22579.044,E2 22579.044} C_VEL
LIN {X 0,Y 584.005,Z 1142.457,A -85,B 0,C 180,E1 22576.939,E2 22576.939} C_VEL
LIN {X 0,Y 584.092,Z 1132.315,A -85,B 0,C 180,E1 22574.817,E2 22574.817} C_VEL
LIN {X 0,Y 584.227,Z 1120.377,A -85,B 0,C 180,E1 22572.675,E2 22572.675} C_VEL
LIN {X 0,Y 584.366,Z 1107.621,A -85,B 0,C 180,E1 22570.717,E2 22570.717} C_VEL
LIN {X 0,Y 584.571,Z 1092.842,A -85,B 0,C 180,E1 22568.739,E2 22568.739} C_VEL
LIN {X 0,Y 584.842,Z 1076.673,A -85,B 0,C 180,E1 22566.845,E2 22566.845} C_VEL
LIN {X 0,Y 585.098,Z 1059.902,A -85,B 0,C 180,E1 22565.141,E2 22565.141} C_VEL
LIN {X 0,Y 585.457,Z 1040.58,A -85,B 0,C 180,E1 22563.42,E2 22563.42} C_VEL
LIN {X 0,Y 585.844,Z 1021.342,A -85,B 0,C 180,E1 22561.928,E2 22561.928} C_VEL
LIN {X 0,Y 586.172,Z 1001.033,A -85,B 0,C 180,E1 22560.577,E2 22560.577} C_VEL
LIN {X 0,Y 586.595,Z 979.662,A -85,B 0,C 180,E1 22559.359,E2 22559.359} C_VEL
LIN {X 0,Y 586.874,Z 959.124,A -85,B 0,C 180,E1 22558.382,E2 22558.382} C_VEL
LIN {X 0,Y 587.252,Z 935.786,A -85,B 0,C 180,E1 22557.476,E2 22557.476} C_VEL
LIN {X 0,Y 587.467,Z 915.237,A -85,B 0,C 180,E1 22556.851,E2 22556.851} C_VEL
LIN {X 0,Y 587.71,Z 891.229,A -85,B 0,C 180,E1 22556.317,E2 22556.317} C_VEL
LIN {X 0,Y 588.478,Z 668.295,A -85,B 0,C 180,E1 22553.072,E2 22553.072} C_VEL
LIN {X 0,Y 588.76,Z 546.64,A -85,B 0,C 180,E1 22551.253,E2 22551.253} C_VEL
LIN {X 0,Y 587.945,Z 541.522,A -85,B 0,C 180,E1 22551.07,E2 22551.07} C_VEL
LIN {X 0,Y 588.14,Z 519.512,A -85,B 0,C 180,E1 22549.681,E2 22549.681} C_VEL
LIN {X 0,Y 584.166,Z 510.752,A -85,B 0,C 180,E1 22548.75,E2 22548.75} C_VEL
LIN {X 0,Y 584.083,Z 510.244,A -85,B 0,C 180,E1 22548.379,E2 22548.379} C_VEL
LIN {X 0,Y 584.077,Z 510.288,A -85,B 0,C 180,E1 22545.13,E2 22545.13} C_VEL
LIN {X 0,Y 584.087,Z 510.289,A -85,B 0,C 180,E1 22542.015,E2 22542.015} C_VEL
LIN {X 0,Y 584.078,Z 510.288,A -85,B 0,C 180,E1 22538.795,E2 22538.795} C_VEL
LIN {X 0,Y 584.084,Z 510.291,A -85,B 0,C 180,E1 22535.593,E2 22535.593} C_VEL
LIN {X 0,Y 584.078,Z 510.283,A -85,B 0,C 180,E1 22532.399,E2 22532.399} C_VEL
LIN {X 0,Y 584.08,Z 510.288,A -85,B 0,C 180,E1 22529.185,E2 22529.185} C_VEL
LIN {X 0,Y 584.078,Z 510.284,A -85,B 0,C 180,E1 22525.991,E2 22525.991} C_VEL
LIN {X 0,Y 584.078,Z 510.284,A -85,B 0,C 180,E1 22522.76,E2 22522.76} C_VEL
LIN {X 0,Y 584.079,Z 510.286,A -85,B 0,C 180,E1 22519.604,E2 22519.604} C_VEL
LIN {X 0,Y 584.078,Z 510.282,A -85,B 0,C 180,E1 22516.407,E2 22516.407} C_VEL
LIN {X 0,Y 584.08,Z 510.285,A -85,B 0,C 180,E1 22513.261,E2 22513.261} C_VEL
LIN {X 0,Y 584.077,Z 510.283,A -85,B 0,C 180,E1 22510.056,E2 22510.056} C_VEL
LIN {X 0,Y 584.081,Z 510.285,A -85,B 0,C 180,E1 22506.843,E2 22506.843} C_VEL
LIN {X 0,Y 584.078,Z 510.285,A -85,B 0,C 180,E1 22503.608,E2 22503.608} C_VEL
LIN {X 0,Y 584.084,Z 510.29,A -85,B 0,C 180,E1 22500.392,E2 22500.392} C_VEL
LIN {X 0,Y 584.079,Z 510.285,A -85,B 0,C 180,E1 22497.154,E2 22497.154} C_VEL
LIN {X 0,Y 584.096,Z 510.294,A -85,B 0,C 180,E1 22493.809,E2 22493.809} C_VEL
LIN {X 0,Y 584.096,Z 510.284,A -85,B 0,C 180,E1 22490.403,E2 22490.403} C_VEL
LIN {X 0,Y 584.083,Z 510.287,A -85,B 0,C 180,E1 22487.142,E2 22487.142} C_VEL
LIN {X 0,Y 584.074,Z 510.283,A -85,B 0,C 180,E1 22486.711,E2 22486.711} C_VEL
LIN {X 0,Y 583.094,Z 510.406,A -85,B 0,C 180,E1 22485.955,E2 22485.955} C_VEL
LIN {X 0,Y 576.677,Z 511.213,A -85,B 0,C 180,E1 22483.835,E2 22483.835} C_VEL
LIN {X 0,Y 576.155,Z 511.283,A -85,B 0,C 180,E1 22483.282,E2 22483.282} C_VEL
LIN {X 0,Y 576.156,Z 511.266,A -85,B 0,C 180,E1 22479.86,E2 22479.86} C_VEL
LIN {X 0,Y 576.141,Z 511.278,A -85,B 0,C 180,E1 22476.583,E2 22476.583} C_VEL
LIN {X 0,Y 576.151,Z 511.27,A -85,B 0,C 180,E1 22473.29,E2 22473.29} C_VEL
LIN {X 0,Y 576.135,Z 511.273,A -85,B 0,C 180,E1 22470.127,E2 22470.127} C_VEL
LIN {X 0,Y 576.149,Z 511.276,A -85,B 0,C 180,E1 22466.862,E2 22466.862} C_VEL
LIN {X 0,Y 576.131,Z 511.277,A -85,B 0,C 180,E1 22463.636,E2 22463.636} C_VEL
LIN {X 0,Y 576.148,Z 511.277,A -85,B 0,C 180,E1 22460.401,E2 22460.401} C_VEL
LIN {X 0,Y 576.13,Z 511.277,A -85,B 0,C 180,E1 22457.232,E2 22457.232} C_VEL
LIN {X 0,Y 576.152,Z 511.282,A -85,B 0,C 180,E1 22453.961,E2 22453.961} C_VEL
LIN {X 0,Y 576.132,Z 511.282,A -85,B 0,C 180,E1 22450.676,E2 22450.676} C_VEL
LIN {X 0,Y 576.193,Z 511.569,A -85,B 0,C 180,E1 22449.705,E2 22449.705} C_VEL
LIN {X 0,Y 578.878,Z 518.076,A -85,B 0,C 180,E1 22448.99,E2 22448.99} C_VEL
LIN {X 0,Y 580.957,Z 522.686,A -85,B 0,C 180,E1 22448.506,E2 22448.506} C_VEL
LIN {X 0,Y 580.215,Z 568.942,A -85,B 0,C 180,E1 22445.442,E2 22445.442} C_VEL
LIN {X 0,Y 580.016,Z 590.435,A -85,B 0,C 180,E1 22444.08,E2 22444.08} C_VEL
LIN {X 0,Y 581.027,Z 597.098,A -85,B 0,C 180,E1 22443.914,E2 22443.914} C_VEL
LIN {X 0,Y 580.111,Z 825.995,A -85,B 0,C 180,E1 22440.687,E2 22440.687} C_VEL
LIN {X 0,Y 579.821,Z 896.717,A -85,B 0,C 180,E1 22439.678,E2 22439.678} C_VEL
LIN {X 0,Y 579.566,Z 917.879,A -85,B 0,C 180,E1 22439.19,E2 22439.19} C_VEL
LIN {X 0,Y 579.229,Z 940.026,A -85,B 0,C 180,E1 22438.491,E2 22438.491} C_VEL
LIN {X 0,Y 578.926,Z 960.573,A -85,B 0,C 180,E1 22437.653,E2 22437.653} C_VEL
LIN {X 0,Y 578.509,Z 980.426,A -85,B 0,C 180,E1 22436.648,E2 22436.648} C_VEL
LIN {X 0,Y 578.086,Z 1000.979,A -85,B 0,C 180,E1 22435.4,E2 22435.4} C_VEL
LIN {X 0,Y 577.706,Z 1019.733,A -85,B 0,C 180,E1 22434.054,E2 22434.054} C_VEL
LIN {X 0,Y 577.306,Z 1037.494,A -85,B 0,C 180,E1 22432.558,E2 22432.558} C_VEL
LIN {X 0,Y 576.952,Z 1053.756,A -85,B 0,C 180,E1 22430.969,E2 22430.969} C_VEL
LIN {X 0,Y 576.652,Z 1070.004,A -85,B 0,C 180,E1 22429.13,E2 22429.13} C_VEL
LIN {X 0,Y 576.436,Z 1083.525,A -85,B 0,C 180,E1 22427.358,E2 22427.358} C_VEL
LIN {X 0,Y 576.238,Z 1095.69,A -85,B 0,C 180,E1 22425.499,E2 22425.499} C_VEL
LIN {X 0,Y 576.092,Z 1107.082,A -85,B 0,C 180,E1 22423.448,E2 22423.448} C_VEL
LIN {X 0,Y 576.005,Z 1116.57,A -85,B 0,C 180,E1 22421.413,E2 22421.413} C_VEL
LIN {X 0,Y 575.943,Z 1124.226,A -85,B 0,C 180,E1 22419.392,E2 22419.392} C_VEL
LIN {X 0,Y 575.908,Z 1130.531,A -85,B 0,C 180,E1 22417.281,E2 22417.281} C_VEL
LIN {X 0,Y 575.902,Z 1135.04,A -85,B 0,C 180,E1 22415.28,E2 22415.28} C_VEL
LIN {X 0,Y 575.908,Z 1138.121,A -85,B 0,C 180,E1 22413.185,E2 22413.185} C_VEL
LIN {X 0,Y 575.91,Z 1139.773,A -85,B 0,C 180,E1 22410.995,E2 22410.995} C_VEL
LIN {X 0,Y 575.911,Z 1139.771,A -85,B 0,C 180,E1 22408.906,E2 22408.906} C_VEL
LIN {X 0,Y 575.908,Z 1138.11,A -85,B 0,C 180,E1 22406.716,E2 22406.716} C_VEL
LIN {X 0,Y 575.903,Z 1135.019,A -85,B 0,C 180,E1 22404.62,E2 22404.62} C_VEL
LIN {X 0,Y 575.908,Z 1130.504,A -85,B 0,C 180,E1 22402.618,E2 22402.618} C_VEL
LIN {X 0,Y 575.942,Z 1123.833,A -85,B 0,C 180,E1 22400.406,E2 22400.406} C_VEL
LIN {X 0,Y 576.008,Z 1116.116,A -85,B 0,C 180,E1 22398.384,E2 22398.384} C_VEL
LIN {X 0,Y 576.096,Z 1106.5,A -85,B 0,C 180,E1 22396.347,E2 22396.347} C_VEL
LIN {X 0,Y 576.24,Z 1094.967,A -85,B 0,C 180,E1 22394.295,E2 22394.295} C_VEL
LIN {X 0,Y 576.445,Z 1082.709,A -85,B 0,C 180,E1 22392.434,E2 22392.434} C_VEL
LIN {X 0,Y 576.698,Z 1068.178,A -85,B 0,C 180,E1 22390.556,E2 22390.556} C_VEL
LIN {X 0,Y 576.971,Z 1053.097,A -85,B 0,C 180,E1 22388.872,E2 22388.872} C_VEL
LIN {X 0,Y 577.326,Z 1036.092,A -85,B 0,C 180,E1 22387.227,E2 22387.227} C_VEL
LIN {X 0,Y 577.739,Z 1018.131,A -85,B 0,C 180,E1 22385.731,E2 22385.731} C_VEL
LIN {X 0,Y 578.145,Z 999.073,A -85,B 0,C 180,E1 22384.383,E2 22384.383} C_VEL
LIN {X 0,Y 578.53,Z 979.06,A -85,B 0,C 180,E1 22383.187,E2 22383.187} C_VEL
LIN {X 0,Y 578.952,Z 958.277,A -85,B 0,C 180,E1 22382.157,E2 22382.157} C_VEL
LIN {X 0,Y 579.284,Z 938.211,A -85,B 0,C 180,E1 22381.353,E2 22381.353} C_VEL
LIN {X 0,Y 579.573,Z 916.677,A -85,B 0,C 180,E1 22380.688,E2 22380.688} C_VEL
LIN {X 0,Y 579.829,Z 895.21,A -85,B 0,C 180,E1 22380.207,E2 22380.207} C_VEL
LIN {X 0,Y 580.726,Z 667.057,A -85,B 0,C 180,E1 22376.992,E2 22376.992} C_VEL
LIN {X 0,Y 580.791,Z 596.537,A -85,B 0,C 180,E1 22375.973,E2 22375.973} C_VEL
LIN {X 0,Y 579.576,Z 590.546,A -85,B 0,C 180,E1 22375.778,E2 22375.778} C_VEL
LIN {X 0,Y 580.203,Z 550.705,A -85,B 0,C 180,E1 22372.656,E2 22372.656} C_VEL
LIN {X 0,Y 580.552,Z 522.319,A -85,B 0,C 180,E1 22370.34,E2 22370.34} C_VEL
LIN {X 0,Y 576.15,Z 511.516,A -85,B 0,C 180,E1 22369.017,E2 22369.017} C_VEL
LIN {X 0,Y 576.099,Z 511.276,A -85,B 0,C 180,E1 22366.172,E2 22366.172} C_VEL
LIN {X 0,Y 576.13,Z 511.261,A -85,B 0,C 180,E1 22362.868,E2 22362.868} C_VEL
LIN {X 0,Y 576.096,Z 511.281,A -85,B 0,C 180,E1 22359.824,E2 22359.824} C_VEL
LIN {X 0,Y 576.129,Z 511.28,A -85,B 0,C 180,E1 22356.531,E2 22356.531} C_VEL
LIN {X 0,Y 576.143,Z 511.529,A -85,B 0,C 180,E1 22354.236,E2 22354.236} C_VEL
LIN {X 0,Y 578.942,Z 520.649,A -85,B 0,C 180,E1 22353.372,E2 22353.372} C_VEL
LIN {X 0,Y 578.767,Z 553.792,A -85,B 0,C 180,E1 22350.84,E2 22350.84} C_VEL
LIN {X 0,Y 578.294,Z 593.389,A -85,B 0,C 180,E1 22347.773,E2 22347.773} C_VEL
LIN {X 0,Y 577.777,Z 636.274,A -85,B 0,C 180,E1 22344.54,E2 22344.54} C_VEL
LIN {X 0,Y 577.31,Z 678.434,A -85,B 0,C 180,E1 22341.435,E2 22341.435} C_VEL
LIN {X 0,Y 577.107,Z 705.497,A -85,B 0,C 180,E1 22339.496,E2 22339.496} C_VEL
LIN {X 0,Y 577.591,Z 712.044,A -85,B 0,C 180,E1 22339.391,E2 22339.391} C_VEL
LIN {X 0,Y 577.253,Z 875.95,A -85,B 0,C 180,E1 22337.271,E2 22337.271} C_VEL
LIN {X 0,Y 577.131,Z 893.617,A -85,B 0,C 180,E1 22336.847,E2 22336.847} C_VEL
LIN {X 0,Y 576.968,Z 910.646,A -85,B 0,C 180,E1 22336.248,E2 22336.248} C_VEL
LIN {X 0,Y 576.794,Z 927.194,A -85,B 0,C 180,E1 22335.46,E2 22335.46} C_VEL
LIN {X 0,Y 576.612,Z 942.674,A -85,B 0,C 180,E1 22334.511,E2 22334.511} C_VEL
LIN {X 0,Y 576.423,Z 957.327,A -85,B 0,C 180,E1 22333.39,E2 22333.39} C_VEL
LIN {X 0,Y 576.275,Z 969.832,A -85,B 0,C 180,E1 22332.221,E2 22332.221} C_VEL
LIN {X 0,Y 576.151,Z 981.415,A -85,B 0,C 180,E1 22330.904,E2 22330.904} C_VEL
LIN {X 0,Y 576.043,Z 992.209,A -85,B 0,C 180,E1 22329.391,E2 22329.391} C_VEL
LIN {X 0,Y 575.979,Z 1001.35,A -85,B 0,C 180,E1 22327.782,E2 22327.782} C_VEL
LIN {X 0,Y 575.941,Z 1008.44,A -85,B 0,C 180,E1 22326.179,E2 22326.179} C_VEL
LIN {X 0,Y 575.92,Z 1013.966,A -85,B 0,C 180,E1 22324.481,E2 22324.481} C_VEL
LIN {X 0,Y 575.913,Z 1017.643,A -85,B 0,C 180,E1 22322.787,E2 22322.787} C_VEL
LIN {X 0,Y 575.914,Z 1019.661,A -85,B 0,C 180,E1 22320.995,E2 22320.995} C_VEL
LIN {X 0,Y 575.916,Z 1019.843,A -85,B 0,C 180,E1 22319.304,E2 22319.304} C_VEL
LIN {X 0,Y 575.911,Z 1018.397,A -85,B 0,C 180,E1 22317.612,E2 22317.612} C_VEL
LIN {X 0,Y 575.915,Z 1015.204,A -85,B 0,C 180,E1 22315.918,E2 22315.918} C_VEL
LIN {X 0,Y 575.933,Z 1010.183,A -85,B 0,C 180,E1 22314.221,E2 22314.221} C_VEL
LIN {X 0,Y 575.963,Z 1003.712,A -85,B 0,C 180,E1 22312.62,E2 22312.62} C_VEL
LIN {X 0,Y 576.021,Z 995.163,A -85,B 0,C 180,E1 22310.996,E2 22310.996} C_VEL
LIN {X 0,Y 576.102,Z 985.918,A -85,B 0,C 180,E1 22309.602,E2 22309.602} C_VEL
LIN {X 0,Y 576.215,Z 975.37,A -85,B 0,C 180,E1 22308.287,E2 22308.287} C_VEL
LIN {X 0,Y 576.371,Z 961.823,A -85,B 0,C 180,E1 22306.916,E2 22306.916} C_VEL
LIN {X 0,Y 576.54,Z 948.247,A -85,B 0,C 180,E1 22305.8,E2 22305.8} C_VEL
LIN {X 0,Y 576.707,Z 933.744,A -85,B 0,C 180,E1 22304.824,E2 22304.824} C_VEL
LIN {X 0,Y 576.884,Z 918.285,A -85,B 0,C 180,E1 22304.004,E2 22304.004} C_VEL
LIN {X 0,Y 577.061,Z 902.24,A -85,B 0,C 180,E1 22303.342,E2 22303.342} C_VEL
LIN {X 0,Y 577.201,Z 884.219,A -85,B 0,C 180,E1 22302.814,E2 22302.814} C_VEL
LIN {X 0,Y 577.282,Z 866.55,A -85,B 0,C 180,E1 22302.493,E2 22302.493} C_VEL
LIN {X 0,Y 577.428,Z 707.784,A -85,B 0,C 180,E1 22300.458,E2 22300.458} C_VEL
LIN {X 0,Y 577.057,Z 704.409,A -85,B 0,C 180,E1 22300.358,E2 22300.358} C_VEL
LIN {X 0,Y 577.53,Z 660.759,A -85,B 0,C 180,E1 22297.182,E2 22297.182} C_VEL
LIN {X 0,Y 578.014,Z 616.211,A -85,B 0,C 180,E1 22293.868,E2 22293.868} C_VEL
LIN {X 0,Y 578.505,Z 574.924,A -85,B 0,C 180,E1 22290.717,E2 22290.717} C_VEL
LIN {X 0,Y 578.893,Z 540.196,A -85,B 0,C 180,E1 22288.037,E2 22288.037} C_VEL
LIN {X 0,Y 578.422,Z 518.944,A -85,B 0,C 180,E1 22286.585,E2 22286.585} C_VEL
LIN {X 0,Y 576.166,Z 511.749,A -85,B 0,C 180,E1 22286.048,E2 22286.048} C_VEL
LIN {X 0,Y 576.105,Z 511.292,A -85,B 0,C 180,E1 22285.88,E2 22285.88} C_VEL
LIN {X 0,Y 576.123,Z 511.28,A -85,B 0,C 180,E1 22282.479,E2 22282.479} C_VEL
LIN {X 0,Y 576.152,Z 511.269,A -85,B 0,C 180,E1 22279.269,E2 22279.269} C_VEL
LIN {X 0,Y 576.143,Z 511.271,A -85,B 0,C 180,E1 22276.039,E2 22276.039} C_VEL
LIN {X 0,Y 576.125,Z 511.254,A -85,B 0,C 180,E1 22272.868,E2 22272.868} C_VEL
LIN {X 0,Y 576.21,Z 511.644,A -85,B 0,C 180,E1 22272.365,E2 22272.365} C_VEL
LIN {X 0,Y 581.256,Z 523.452,A -85,B 0,C 180,E1 22270.949,E2 22270.949} C_VEL
LIN {X 0,Y 581.035,Z 543.928,A -85,B 0,C 180,E1 22269.408,E2 22269.408} C_VEL
LIN {X 0,Y 582.647,Z 551.792,A -85,B 0,C 180,E1 22269.151,E2 22269.151} C_VEL
LIN {X 0,Y 581.666,Z 759.267,A -85,B 0,C 180,E1 22266.06,E2 22266.06} C_VEL
LIN {X 0,Y 581.041,Z 891.761,A -85,B 0,C 180,E1 22264.113,E2 22264.113} C_VEL
LIN {X 0,Y 580.713,Z 915.594,A -85,B 0,C 180,E1 22263.575,E2 22263.575} C_VEL
LIN {X 0,Y 580.416,Z 936.939,A -85,B 0,C 180,E1 22262.916,E2 22262.916} C_VEL
LIN {X 0,Y 579.921,Z 959.677,A -85,B 0,C 180,E1 22262.017,E2 22262.017} C_VEL
LIN {X 0,Y 579.518,Z 981.394,A -85,B 0,C 180,E1 22260.965,E2 22260.965} C_VEL
LIN {X 0,Y 578.967,Z 1001.927,A -85,B 0,C 180,E1 22259.769,E2 22259.769} C_VEL
LIN {X 0,Y 578.481,Z 1023.144,A -85,B 0,C 180,E1 22258.324,E2 22258.324} C_VEL
LIN {X 0,Y 577.996,Z 1041.906,A -85,B 0,C 180,E1 22256.84,E2 22256.84} C_VEL
LIN {X 0,Y 577.555,Z 1059.902,A -85,B 0,C 180,E1 22255.206,E2 22255.206} C_VEL
LIN {X 0,Y 577.18,Z 1076.97,A -85,B 0,C 180,E1 22253.447,E2 22253.447} C_VEL
LIN {X 0,Y 576.818,Z 1092.842,A -85,B 0,C 180,E1 22251.561,E2 22251.561} C_VEL
LIN {X 0,Y 576.528,Z 1108.332,A -85,B 0,C 180,E1 22249.45,E2 22249.45} C_VEL
LIN {X 0,Y 576.328,Z 1121.643,A -85,B 0,C 180,E1 22247.362,E2 22247.362} C_VEL
LIN {X 0,Y 576.151,Z 1133.165,A -85,B 0,C 180,E1 22245.23,E2 22245.23} C_VEL
LIN {X 0,Y 576.037,Z 1143.288,A -85,B 0,C 180,E1 22243.041,E2 22243.041} C_VEL
LIN {X 0,Y 575.967,Z 1151.051,A -85,B 0,C 180,E1 22241.009,E2 22241.009} C_VEL
LIN {X 0,Y 575.943,Z 1158.04,A -85,B 0,C 180,E1 22238.788,E2 22238.788} C_VEL
LIN {X 0,Y 575.916,Z 1163.254,A -85,B 0,C 180,E1 22236.58,E2 22236.58} C_VEL
LIN {X 0,Y 575.914,Z 1167.163,A -85,B 0,C 180,E1 22234.281,E2 22234.281} C_VEL
LIN {X 0,Y 575.914,Z 1169.256,A -85,B 0,C 180,E1 22232.089,E2 22232.089} C_VEL
LIN {X 0,Y 575.899,Z 1169.962,A -85,B 0,C 180,E1 22229.801,E2 22229.801} C_VEL
LIN {X 0,Y 575.916,Z 1169.122,A -85,B 0,C 180,E1 22227.712,E2 22227.712} C_VEL
LIN {X 0,Y 575.904,Z 1166.753,A -85,B 0,C 180,E1 22225.419,E2 22225.419} C_VEL
LIN {X 0,Y 575.903,Z 1162.909,A -85,B 0,C 180,E1 22223.253,E2 22223.253} C_VEL
LIN {X 0,Y 575.947,Z 1157.475,A -85,B 0,C 180,E1 22221.011,E2 22221.011} C_VEL
LIN {X 0,Y 575.966,Z 1150.694,A -85,B 0,C 180,E1 22218.89,E2 22218.89} C_VEL
LIN {X 0,Y 576.037,Z 1142.456,A -85,B 0,C 180,E1 22216.755,E2 22216.755} C_VEL
LIN {X 0,Y 576.152,Z 1132.317,A -85,B 0,C 180,E1 22214.602,E2 22214.602} C_VEL
LIN {X 0,Y 576.337,Z 1120.375,A -85,B 0,C 180,E1 22212.43,E2 22212.43} C_VEL
LIN {X 0,Y 576.546,Z 1107.623,A -85,B 0,C 180,E1 22210.445,E2 22210.445} C_VEL
LIN {X 0,Y 576.818,Z 1092.843,A -85,B 0,C 180,E1 22208.44,E2 22208.44} C_VEL
LIN {X 0,Y 577.187,Z 1076.673,A -85,B 0,C 180,E1 22206.52,E2 22206.52} C_VEL
LIN {X 0,Y 577.574,Z 1059.35,A -85,B 0,C 180,E1 22204.74,E2 22204.74} C_VEL
LIN {X 0,Y 578.039,Z 1039.678,A -85,B 0,C 180,E1 22202.975,E2 22202.975} C_VEL
LIN {X 0,Y 578.575,Z 1020.185,A -85,B 0,C 180,E1 22201.456,E2 22201.456} C_VEL
LIN {X 0,Y 579.038,Z 999.691,A -85,B 0,C 180,E1 22200.092,E2 22200.092} C_VEL
LIN {X 0,Y 579.567,Z 977.429,A -85,B 0,C 180,E1 22198.831,E2 22198.831} C_VEL
LIN {X 0,Y 580.001,Z 956.994,A -85,B 0,C 180,E1 22197.865,E2 22197.865} C_VEL
LIN {X 0,Y 580.441,Z 934.174,A -85,B 0,C 180,E1 22196.991,E2 22196.991} C_VEL
LIN {X 0,Y 580.75,Z 913.281,A -85,B 0,C 180,E1 22196.362,E2 22196.362} C_VEL
LIN {X 0,Y 581.048,Z 890.179,A -85,B 0,C 180,E1 22195.86,E2 22195.86} C_VEL
LIN {X 0,Y 582.073,Z 669.567,A -85,B 0,C 180,E1 22192.616,E2 22192.616} C_VEL
LIN {X 0,Y 582.508,Z 548.335,A -85,B 0,C 180,E1 22190.784,E2 22190.784} C_VEL
LIN {X 0,Y 581.372,Z 541.629,A -85,B 0,C 180,E1 22190.551,E2 22190.551} C_VEL
LIN {X 0,Y 581.604,Z 523.215,A -85,B 0,C 180,E1 22189.376,E2 22189.376} C_VEL
LIN {X 0,Y 576.22,Z 511.75,A -85,B 0,C 180,E1 22188.123,E2 22188.123} C_VEL
LIN {X 0,Y 576.147,Z 511.235,A -85,B 0,C 180,E1 22187.808,E2 22187.808} C_VEL
LIN {X 0,Y 576.152,Z 511.268,A -85,B 0,C 180,E1 22184.5,E2 22184.5} C_VEL
LIN {X 0,Y 576.15,Z 511.27,A -85,B 0,C 180,E1 22181.126,E2 22181.126} C_VEL
LIN {X 0,Y 576.149,Z 511.274,A -85,B 0,C 180,E1 22177.85,E2 22177.85} C_VEL
LIN {X 0,Y 576.142,Z 511.276,A -85,B 0,C 180,E1 22174.575,E2 22174.575} C_VEL
LIN {X 0,Y 576.143,Z 511.279,A -85,B 0,C 180,E1 22171.368,E2 22171.368} C_VEL
LIN {X 0,Y 576.14,Z 511.274,A -85,B 0,C 180,E1 22168.163,E2 22168.163} C_VEL
LIN {X 0,Y 576.141,Z 511.279,A -85,B 0,C 180,E1 22164.942,E2 22164.942} C_VEL
LIN {X 0,Y 576.14,Z 511.271,A -85,B 0,C 180,E1 22161.694,E2 22161.694} C_VEL
LIN {X 0,Y 576.143,Z 511.276,A -85,B 0,C 180,E1 22158.412,E2 22158.412} C_VEL
LIN {X 0,Y 576.142,Z 511.271,A -85,B 0,C 180,E1 22155.191,E2 22155.191} C_VEL
LIN {X 0,Y 576.145,Z 511.274,A -85,B 0,C 180,E1 22151.918,E2 22151.918} C_VEL
LIN {X 0,Y 576.155,Z 511.271,A -85,B 0,C 180,E1 22148.583,E2 22148.583} C_VEL
LIN {X 0,Y 576.154,Z 511.273,A -85,B 0,C 180,E1 22145.177,E2 22145.177} C_VEL
LIN {X 0,Y 576.144,Z 511.28,A -85,B 0,C 180,E1 22141.889,E2 22141.889} C_VEL
LIN {X 0,Y 576.146,Z 511.275,A -85,B 0,C 180,E1 22138.608,E2 22138.608} C_VEL
LIN {X 0,Y 576.138,Z 511.279,A -85,B 0,C 180,E1 22135.421,E2 22135.421} C_VEL
LIN {X 0,Y 576.145,Z 511.273,A -85,B 0,C 180,E1 22132.22,E2 22132.22} C_VEL
LIN {X 0,Y 576.134,Z 511.273,A -85,B 0,C 180,E1 22128.994,E2 22128.994} C_VEL
LIN {X 0,Y 576.144,Z 511.272,A -85,B 0,C 180,E1 22125.733,E2 22125.733} C_VEL
LIN {X 0,Y 576.155,Z 511.283,A -85,B 0,C 180,E1 22123.282,E2 22123.282} C_VEL
LIN {X 0,Y 575.184,Z 511.409,A -85,B 0,C 180,E1 22122.516,E2 22122.516} C_VEL
LIN {X 0,Y 568.664,Z 512.199,A -85,B 0,C 180,E1 22120.311,E2 22120.311} C_VEL
LIN {X 0,Y 568.216,Z 512.254,A -85,B 0,C 180,E1 22119.806,E2 22119.806} C_VEL
LIN {X 0,Y 568.198,Z 512.265,A -85,B 0,C 180,E1 22116.464,E2 22116.464} C_VEL
LIN {X 0,Y 568.209,Z 512.26,A -85,B 0,C 180,E1 22113.145,E2 22113.145} C_VEL
LIN {X 0,Y 568.193,Z 512.259,A -85,B 0,C 180,E1 22109.972,E2 22109.972} C_VEL
LIN {X 0,Y 568.21,Z 512.267,A -85,B 0,C 180,E1 22106.7,E2 22106.7} C_VEL
LIN {X 0,Y 568.192,Z 512.265,A -85,B 0,C 180,E1 22103.502,E2 22103.502} C_VEL
LIN {X 0,Y 568.211,Z 512.263,A -85,B 0,C 180,E1 22100.262,E2 22100.262} C_VEL
LIN {X 0,Y 568.193,Z 512.264,A -85,B 0,C 180,E1 22097.058,E2 22097.058} C_VEL
LIN {X 0,Y 568.216,Z 512.266,A -85,B 0,C 180,E1 22093.752,E2 22093.752} C_VEL
LIN {X 0,Y 568.209,Z 512.309,A -85,B 0,C 180,E1 22090.49,E2 22090.49} C_VEL
LIN {X 0,Y 568.301,Z 512.8,A -85,B 0,C 180,E1 22090.259,E2 22090.259} C_VEL
LIN {X 0,Y 574.246,Z 526.436,A -85,B 0,C 180,E1 22088.779,E2 22088.779} C_VEL
LIN {X 0,Y 573.307,Z 573.533,A -85,B 0,C 180,E1 22085.627,E2 22085.627} C_VEL
LIN {X 0,Y 573.089,Z 590.353,A -85,B 0,C 180,E1 22084.553,E2 22084.553} C_VEL
LIN {X 0,Y 574.382,Z 598.505,A -85,B 0,C 180,E1 22084.34,E2 22084.34} C_VEL
LIN {X 0,Y 573.224,Z 827.898,A -85,B 0,C 180,E1 22081.07,E2 22081.07} C_VEL
LIN {X 0,Y 572.866,Z 896.758,A -85,B 0,C 180,E1 22080.075,E2 22080.075} C_VEL
LIN {X 0,Y 572.543,Z 918.094,A -85,B 0,C 180,E1 22079.578,E2 22079.578} C_VEL
LIN {X 0,Y 572.132,Z 940.309,A -85,B 0,C 180,E1 22078.867,E2 22078.867} C_VEL
LIN {X 0,Y 571.726,Z 961.245,A -85,B 0,C 180,E1 22078,E2 22078} C_VEL
LIN {X 0,Y 571.198,Z 981.436,A -85,B 0,C 180,E1 22076.96,E2 22076.96} C_VEL
LIN {X 0,Y 570.668,Z 1001.795,A -85,B 0,C 180,E1 22075.699,E2 22075.699} C_VEL
LIN {X 0,Y 570.164,Z 1020.841,A -85,B 0,C 180,E1 22074.301,E2 22074.301} C_VEL
LIN {X 0,Y 569.674,Z 1038.71,A -85,B 0,C 180,E1 22072.769,E2 22072.769} C_VEL
LIN {X 0,Y 569.217,Z 1055.281,A -85,B 0,C 180,E1 22071.106,E2 22071.106} C_VEL
LIN {X 0,Y 568.845,Z 1070.946,A -85,B 0,C 180,E1 22069.285,E2 22069.285} C_VEL
LIN {X 0,Y 568.55,Z 1084.944,A -85,B 0,C 180,E1 22067.395,E2 22067.395} C_VEL
LIN {X 0,Y 568.318,Z 1097.591,A -85,B 0,C 180,E1 22065.406,E2 22065.406} C_VEL
LIN {X 0,Y 568.138,Z 1108.644,A -85,B 0,C 180,E1 22063.329,E2 22063.329} C_VEL
LIN {X 0,Y 568.025,Z 1118.204,A -85,B 0,C 180,E1 22061.165,E2 22061.165} C_VEL
LIN {X 0,Y 567.961,Z 1125.611,A -85,B 0,C 180,E1 22059.116,E2 22059.116} C_VEL
LIN {X 0,Y 567.914,Z 1131.295,A -85,B 0,C 180,E1 22057.079,E2 22057.079} C_VEL
LIN {X 0,Y 567.895,Z 1135.894,A -85,B 0,C 180,E1 22054.848,E2 22054.848} C_VEL
LIN {X 0,Y 567.892,Z 1138.683,A -85,B 0,C 180,E1 22052.725,E2 22052.725} C_VEL
LIN {X 0,Y 567.895,Z 1139.862,A -85,B 0,C 180,E1 22050.605,E2 22050.605} C_VEL
LIN {X 0,Y 567.9,Z 1139.611,A -85,B 0,C 180,E1 22048.487,E2 22048.487} C_VEL
LIN {X 0,Y 567.907,Z 1137.773,A -85,B 0,C 180,E1 22046.366,E2 22046.366} C_VEL
LIN {X 0,Y 567.919,Z 1134.136,A -85,B 0,C 180,E1 22044.11,E2 22044.11} C_VEL
LIN {X 0,Y 567.95,Z 1129.216,A -85,B 0,C 180,E1 22042.005,E2 22042.005} C_VEL
LIN {X 0,Y 567.986,Z 1122.411,A -85,B 0,C 180,E1 22039.861,E2 22039.861} C_VEL
LIN {X 0,Y 568.074,Z 1113.59,A -85,B 0,C 180,E1 22037.647,E2 22037.647} C_VEL
LIN {X 0,Y 568.215,Z 1103.871,A -85,B 0,C 180,E1 22035.634,E2 22035.634} C_VEL
LIN {X 0,Y 568.401,Z 1092.399,A -85,B 0,C 180,E1 22033.653,E2 22033.653} C_VEL
LIN {X 0,Y 568.667,Z 1078.838,A -85,B 0,C 180,E1 22031.656,E2 22031.656} C_VEL
LIN {X 0,Y 569.004,Z 1063.949,A -85,B 0,C 180,E1 22029.777,E2 22029.777} C_VEL
LIN {X 0,Y 569.42,Z 1048.51,A -85,B 0,C 180,E1 22028.091,E2 22028.091} C_VEL
LIN {X 0,Y 569.868,Z 1031.449,A -85,B 0,C 180,E1 22026.493,E2 22026.493} C_VEL
LIN {X 0,Y 570.368,Z 1012.907,A -85,B 0,C 180,E1 22025,E2 22025} C_VEL
LIN {X 0,Y 570.893,Z 993.074,A -85,B 0,C 180,E1 22023.642,E2 22023.642} C_VEL
LIN {X 0,Y 571.433,Z 973.017,A -85,B 0,C 180,E1 22022.488,E2 22022.488} C_VEL
LIN {X 0,Y 571.892,Z 952.414,A -85,B 0,C 180,E1 22021.522,E2 22021.522} C_VEL
LIN {X 0,Y 572.332,Z 930.697,A -85,B 0,C 180,E1 22020.711,E2 22020.711} C_VEL
LIN {X 0,Y 572.703,Z 909.332,A -85,B 0,C 180,E1 22020.103,E2 22020.103} C_VEL
LIN {X 0,Y 572.92,Z 888.069,A -85,B 0,C 180,E1 22019.691,E2 22019.691} C_VEL
LIN {X 0,Y 574.02,Z 666.134,A -85,B 0,C 180,E1 22016.544,E2 22016.544} C_VEL
LIN {X 0,Y 574.179,Z 598.305,A -85,B 0,C 180,E1 22015.553,E2 22015.553} C_VEL
LIN {X 0,Y 572.571,Z 590.551,A -85,B 0,C 180,E1 22015.3,E2 22015.3} C_VEL
LIN {X 0,Y 573.372,Z 550.695,A -85,B 0,C 180,E1 22012.133,E2 22012.133} C_VEL
LIN {X 0,Y 573.854,Z 526.242,A -85,B 0,C 180,E1 22010.119,E2 22010.119} C_VEL
LIN {X 0,Y 569.116,Z 515.183,A -85,B 0,C 180,E1 22008.759,E2 22008.759} C_VEL
LIN {X 0,Y 568.18,Z 512.416,A -85,B 0,C 180,E1 22008.37,E2 22008.37} C_VEL
LIN {X 0,Y 568.216,Z 512.27,A -85,B 0,C 180,E1 22005.165,E2 22005.165} C_VEL
LIN {X 0,Y 568.154,Z 512.251,A -85,B 0,C 180,E1 22002.042,E2 22002.042} C_VEL
LIN {X 0,Y 568.208,Z 512.269,A -85,B 0,C 180,E1 21998.782,E2 21998.782} C_VEL
LIN {X 0,Y 568.151,Z 512.267,A -85,B 0,C 180,E1 21995.752,E2 21995.752} C_VEL
LIN {X 0,Y 568.244,Z 512.509,A -85,B 0,C 180,E1 21994.589,E2 21994.589} C_VEL
LIN {X 0,Y 571.551,Z 523.214,A -85,B 0,C 180,E1 21993.56,E2 21993.56} C_VEL
LIN {X 0,Y 571.331,Z 560.231,A -85,B 0,C 180,E1 21990.732,E2 21990.732} C_VEL
LIN {X 0,Y 570.943,Z 592.671,A -85,B 0,C 180,E1 21988.219,E2 21988.219} C_VEL
LIN {X 0,Y 570.297,Z 635.555,A -85,B 0,C 180,E1 21984.939,E2 21984.939} C_VEL
LIN {X 0,Y 569.718,Z 676.99,A -85,B 0,C 180,E1 21981.843,E2 21981.843} C_VEL
LIN {X 0,Y 569.449,Z 705.66,A -85,B 0,C 180,E1 21979.766,E2 21979.766} C_VEL
LIN {X 0,Y 570.046,Z 712.504,A -85,B 0,C 180,E1 21979.653,E2 21979.653} C_VEL
LIN {X 0,Y 569.611,Z 875.991,A -85,B 0,C 180,E1 21977.51,E2 21977.51} C_VEL
LIN {X 0,Y 569.457,Z 893.634,A -85,B 0,C 180,E1 21977.081,E2 21977.081} C_VEL
LIN {X 0,Y 569.25,Z 911.029,A -85,B 0,C 180,E1 21976.458,E2 21976.458} C_VEL
LIN {X 0,Y 569.044,Z 926.778,A -85,B 0,C 180,E1 21975.7,E2 21975.7} C_VEL
LIN {X 0,Y 568.816,Z 941.958,A -85,B 0,C 180,E1 21974.767,E2 21974.767} C_VEL
LIN {X 0,Y 568.578,Z 956.736,A -85,B 0,C 180,E1 21973.63,E2 21973.63} C_VEL
LIN {X 0,Y 568.375,Z 969.836,A -85,B 0,C 180,E1 21972.393,E2 21972.393} C_VEL
LIN {X 0,Y 568.216,Z 981.421,A -85,B 0,C 180,E1 21971.058,E2 21971.058} C_VEL
LIN {X 0,Y 568.084,Z 992.216,A -85,B 0,C 180,E1 21969.523,E2 21969.523} C_VEL
LIN {X 0,Y 567.996,Z 1001.353,A -85,B 0,C 180,E1 21967.892,E2 21967.892} C_VEL
LIN {X 0,Y 567.948,Z 1008.44,A -85,B 0,C 180,E1 21966.267,E2 21966.267} C_VEL
LIN {X 0,Y 567.922,Z 1013.968,A -85,B 0,C 180,E1 21964.544,E2 21964.544} C_VEL
LIN {X 0,Y 567.914,Z 1017.646,A -85,B 0,C 180,E1 21962.826,E2 21962.826} C_VEL
LIN {X 0,Y 567.915,Z 1019.663,A -85,B 0,C 180,E1 21961.009,E2 21961.009} C_VEL
LIN {X 0,Y 567.916,Z 1019.835,A -85,B 0,C 180,E1 21959.294,E2 21959.294} C_VEL
LIN {X 0,Y 567.912,Z 1018.395,A -85,B 0,C 180,E1 21957.579,E2 21957.579} C_VEL
LIN {X 0,Y 567.916,Z 1015.203,A -85,B 0,C 180,E1 21955.861,E2 21955.861} C_VEL
LIN {X 0,Y 567.937,Z 1010.525,A -85,B 0,C 180,E1 21954.241,E2 21954.241} C_VEL
LIN {X 0,Y 567.974,Z 1004.171,A -85,B 0,C 180,E1 21952.617,E2 21952.617} C_VEL
LIN {X 0,Y 568.053,Z 995.259,A -85,B 0,C 180,E1 21950.885,E2 21950.885} C_VEL
LIN {X 0,Y 568.155,Z 985.904,A -85,B 0,C 180,E1 21949.454,E2 21949.454} C_VEL
LIN {X 0,Y 568.299,Z 975.36,A -85,B 0,C 180,E1 21948.121,E2 21948.121} C_VEL
LIN {X 0,Y 568.502,Z 961.631,A -85,B 0,C 180,E1 21946.715,E2 21946.715} C_VEL
LIN {X 0,Y 568.713,Z 948.167,A -85,B 0,C 180,E1 21945.596,E2 21945.596} C_VEL
LIN {X 0,Y 568.926,Z 933.735,A -85,B 0,C 180,E1 21944.611,E2 21944.611} C_VEL
LIN {X 0,Y 569.154,Z 917.469,A -85,B 0,C 180,E1 21943.744,E2 21943.744} C_VEL
LIN {X 0,Y 569.378,Z 901.42,A -85,B 0,C 180,E1 21943.081,E2 21943.081} C_VEL
LIN {X 0,Y 569.547,Z 883.924,A -85,B 0,C 180,E1 21942.57,E2 21942.57} C_VEL
LIN {X 0,Y 569.65,Z 866.257,A -85,B 0,C 180,E1 21942.248,E2 21942.248} C_VEL
LIN {X 0,Y 569.869,Z 708.628,A -85,B 0,C 180,E1 21940.2,E2 21940.2} C_VEL
LIN {X 0,Y 569.384,Z 704.399,A -85,B 0,C 180,E1 21940.083,E2 21940.083} C_VEL
LIN {X 0,Y 569.974,Z 660.749,A -85,B 0,C 180,E1 21936.863,E2 21936.863} C_VEL
LIN {X 0,Y 570.58,Z 616.451,A -85,B 0,C 180,E1 21933.52,E2 21933.52} C_VEL
LIN {X 0,Y 571.236,Z 574.914,A -85,B 0,C 180,E1 21930.308,E2 21930.308} C_VEL
LIN {X 0,Y 571.246,Z 556.261,A -85,B 0,C 180,E1 21928.913,E2 21928.913} C_VEL
LIN {X 0,Y 570.906,Z 529.301,A -85,B 0,C 180,E1 21927.058,E2 21927.058} C_VEL
LIN {X 0,Y 570.41,Z 520.605,A -85,B 0,C 180,E1 21926.485,E2 21926.485} C_VEL
LIN {X 0,Y 568.213,Z 512.604,A -85,B 0,C 180,E1 21925.886,E2 21925.886} C_VEL
LIN {X 0,Y 568.219,Z 512.272,A -85,B 0,C 180,E1 21925.364,E2 21925.364} C_VEL
LIN {X 0,Y 568.179,Z 512.271,A -85,B 0,C 180,E1 21922.11,E2 21922.11} C_VEL
LIN {X 0,Y 568.217,Z 512.261,A -85,B 0,C 180,E1 21918.845,E2 21918.845} C_VEL
LIN {X 0,Y 568.208,Z 512.255,A -85,B 0,C 180,E1 21915.453,E2 21915.453} C_VEL
LIN {X 0,Y 568.221,Z 512.497,A -85,B 0,C 180,E1 21913.053,E2 21913.053} C_VEL
LIN {X 0,Y 569.44,Z 515.622,A -85,B 0,C 180,E1 21912.634,E2 21912.634} C_VEL
LIN {X 0,Y 574.611,Z 527.582,A -85,B 0,C 180,E1 21911.195,E2 21911.195} C_VEL
LIN {X 0,Y 574.376,Z 543.849,A -85,B 0,C 180,E1 21909.959,E2 21909.959} C_VEL
LIN {X 0,Y 576.427,Z 553.632,A -85,B 0,C 180,E1 21909.627,E2 21909.627} C_VEL
LIN {X 0,Y 575.183,Z 761.303,A -85,B 0,C 180,E1 21906.501,E2 21906.501} C_VEL
LIN {X 0,Y 574.408,Z 891.868,A -85,B 0,C 180,E1 21904.56,E2 21904.56} C_VEL
LIN {X 0,Y 573.997,Z 915.62,A -85,B 0,C 180,E1 21904.02,E2 21904.02} C_VEL
LIN {X 0,Y 573.618,Z 937.298,A -85,B 0,C 180,E1 21903.344,E2 21903.344} C_VEL
LIN {X 0,Y 573.022,Z 959.68,A -85,B 0,C 180,E1 21902.45,E2 21902.45} C_VEL
LIN {X 0,Y 572.504,Z 980.783,A -85,B 0,C 180,E1 21901.421,E2 21901.421} C_VEL
LIN {X 0,Y 571.825,Z 1001.93,A -85,B 0,C 180,E1 21900.179,E2 21900.179} C_VEL
LIN {X 0,Y 571.197,Z 1023.113,A -85,B 0,C 180,E1 21898.721,E2 21898.721} C_VEL
LIN {X 0,Y 570.578,Z 1041.908,A -85,B 0,C 180,E1 21897.217,E2 21897.217} C_VEL
LIN {X 0,Y 570.011,Z 1060.456,A -85,B 0,C 180,E1 21895.508,E2 21895.508} C_VEL
LIN {X 0,Y 569.516,Z 1077.615,A -85,B 0,C 180,E1 21893.706,E2 21893.706} C_VEL
LIN {X 0,Y 569.063,Z 1093.692,A -85,B 0,C 180,E1 21891.761,E2 21891.761} C_VEL
LIN {X 0,Y 568.715,Z 1108.333,A -85,B 0,C 180,E1 21889.728,E2 21889.728} C_VEL
LIN {X 0,Y 568.447,Z 1121.008,A -85,B 0,C 180,E1 21887.716,E2 21887.716} C_VEL
LIN {X 0,Y 568.221,Z 1132.317,A -85,B 0,C 180,E1 21885.618,E2 21885.618} C_VEL
LIN {X 0,Y 568.075,Z 1142.455,A -85,B 0,C 180,E1 21883.434,E2 21883.434} C_VEL
LIN {X 0,Y 567.988,Z 1150.695,A -85,B 0,C 180,E1 21881.268,E2 21881.268} C_VEL
LIN {X 0,Y 567.954,Z 1157.475,A -85,B 0,C 180,E1 21879.116,E2 21879.116} C_VEL
LIN {X 0,Y 567.899,Z 1162.84,A -85,B 0,C 180,E1 21876.876,E2 21876.876} C_VEL
LIN {X 0,Y 567.904,Z 1166.594,A -85,B 0,C 180,E1 21874.747,E2 21874.747} C_VEL
LIN {X 0,Y 567.915,Z 1169.055,A -85,B 0,C 180,E1 21872.422,E2 21872.422} C_VEL
LIN {X 0,Y 567.892,Z 1169.939,A -85,B 0,C 180,E1 21870.303,E2 21870.303} C_VEL
LIN {X 0,Y 567.91,Z 1169.323,A -85,B 0,C 180,E1 21867.982,E2 21867.982} C_VEL
LIN {X 0,Y 567.916,Z 1167.276,A -85,B 0,C 180,E1 21865.759,E2 21865.759} C_VEL
LIN {X 0,Y 567.918,Z 1163.46,A -85,B 0,C 180,E1 21863.429,E2 21863.429} C_VEL
LIN {X 0,Y 567.948,Z 1158.55,A -85,B 0,C 180,E1 21861.292,E2 21861.292} C_VEL
LIN {X 0,Y 567.984,Z 1151.764,A -85,B 0,C 180,E1 21859.04,E2 21859.04} C_VEL
LIN {X 0,Y 568.066,Z 1144.108,A -85,B 0,C 180,E1 21856.98,E2 21856.98} C_VEL
LIN {X 0,Y 568.211,Z 1133.61,A -85,B 0,C 180,E1 21854.641,E2 21854.641} C_VEL
LIN {X 0,Y 568.43,Z 1122.237,A -85,B 0,C 180,E1 21852.495,E2 21852.495} C_VEL
LIN {X 0,Y 568.694,Z 1109.042,A -85,B 0,C 180,E1 21850.378,E2 21850.378} C_VEL
LIN {X 0,Y 569.044,Z 1094.537,A -85,B 0,C 180,E1 21848.347,E2 21848.347} C_VEL
LIN {X 0,Y 569.45,Z 1079.476,A -85,B 0,C 180,E1 21846.511,E2 21846.511} C_VEL
LIN {X 0,Y 569.95,Z 1062.115,A -85,B 0,C 180,E1 21844.656,E2 21844.656} C_VEL
LIN {X 0,Y 570.535,Z 1043.892,A -85,B 0,C 180,E1 21842.95,E2 21842.95} C_VEL
LIN {X 0,Y 571.14,Z 1024.608,A -85,B 0,C 180,E1 21841.393,E2 21841.393} C_VEL
LIN {X 0,Y 571.765,Z 1003.711,A -85,B 0,C 180,E1 21839.933,E2 21839.933} C_VEL
LIN {X 0,Y 572.4,Z 983.829,A -85,B 0,C 180,E1 21838.748,E2 21838.748} C_VEL
LIN {X 0,Y 572.972,Z 961.418,A -85,B 0,C 180,E1 21837.628,E2 21837.628} C_VEL
LIN {X 0,Y 573.582,Z 939.362,A -85,B 0,C 180,E1 21836.727,E2 21836.727} C_VEL
LIN {X 0,Y 573.983,Z 916.823,A -85,B 0,C 180,E1 21836.013,E2 21836.013} C_VEL
LIN {X 0,Y 574.392,Z 893.905,A -85,B 0,C 180,E1 21835.475,E2 21835.475} C_VEL
LIN {X 0,Y 574.754,Z 837.94,A -85,B 0,C 180,E1 21834.626,E2 21834.626} C_VEL
LIN {X 0,Y 575.958,Z 629.515,A -85,B 0,C 180,E1 21831.528,E2 21831.528} C_VEL
LIN {X 0,Y 576.287,Z 549.969,A -85,B 0,C 180,E1 21830.303,E2 21830.303} C_VEL
LIN {X 0,Y 574.851,Z 542.193,A -85,B 0,C 180,E1 21830.048,E2 21830.048} C_VEL
LIN {X 0,Y 575.019,Z 527.116,A -85,B 0,C 180,E1 21829.07,E2 21829.07} C_VEL
LIN {X 0,Y 569.494,Z 515.677,A -85,B 0,C 180,E1 21827.808,E2 21827.808} C_VEL
LIN {X 0,Y 568.24,Z 512.496,A -85,B 0,C 180,E1 21827.423,E2 21827.423} C_VEL
LIN {X 0,Y 568.21,Z 512.256,A -85,B 0,C 180,E1 21824.172,E2 21824.172} C_VEL
LIN {X 0,Y 568.199,Z 512.259,A -85,B 0,C 180,E1 21820.889,E2 21820.889} C_VEL
LIN {X 0,Y 568.204,Z 512.259,A -85,B 0,C 180,E1 21817.633,E2 21817.633} C_VEL
LIN {X 0,Y 568.199,Z 512.268,A -85,B 0,C 180,E1 21814.381,E2 21814.381} C_VEL
LIN {X 0,Y 568.205,Z 512.266,A -85,B 0,C 180,E1 21811.154,E2 21811.154} C_VEL
LIN {X 0,Y 568.202,Z 512.265,A -85,B 0,C 180,E1 21807.909,E2 21807.909} C_VEL
LIN {X 0,Y 568.207,Z 512.265,A -85,B 0,C 180,E1 21804.648,E2 21804.648} C_VEL
LIN {X 0,Y 568.214,Z 512.259,A -85,B 0,C 180,E1 21801.253,E2 21801.253} C_VEL
LIN {X 0,Y 568.212,Z 512.263,A -85,B 0,C 180,E1 21797.828,E2 21797.828} C_VEL
LIN {X 0,Y 568.205,Z 512.263,A -85,B 0,C 180,E1 21794.573,E2 21794.573} C_VEL
LIN {X 0,Y 568.204,Z 512.265,A -85,B 0,C 180,E1 21791.263,E2 21791.263} C_VEL
LIN {X 0,Y 568.199,Z 512.26,A -85,B 0,C 180,E1 21787.991,E2 21787.991} C_VEL
LIN {X 0,Y 568.205,Z 512.267,A -85,B 0,C 180,E1 21784.744,E2 21784.744} C_VEL
LIN {X 0,Y 568.199,Z 512.266,A -85,B 0,C 180,E1 21781.512,E2 21781.512} C_VEL
LIN {X 0,Y 568.207,Z 512.267,A -85,B 0,C 180,E1 21778.286,E2 21778.286} C_VEL
LIN {X 0,Y 568.208,Z 512.263,A -85,B 0,C 180,E1 21774.952,E2 21774.952} C_VEL
LIN {X 0,Y 568.213,Z 512.272,A -85,B 0,C 180,E1 21771.5,E2 21771.5} C_VEL
LIN {X 0,Y 568.211,Z 512.257,A -85,B 0,C 180,E1 21768.119,E2 21768.119} C_VEL
LIN {X 0,Y 568.2,Z 512.269,A -85,B 0,C 180,E1 21764.904,E2 21764.904} C_VEL
LIN {X 0,Y 568.208,Z 512.261,A -85,B 0,C 180,E1 21761.64,E2 21761.64} C_VEL
LIN {X 0,Y 568.216,Z 512.254,A -85,B 0,C 180,E1 21759.806,E2 21759.806} C_VEL
LIN {X 0,Y 567.211,Z 512.391,A -85,B 0,C 180,E1 21759.03,E2 21759.03} C_VEL
LIN {X 0,Y 560.782,Z 513.195,A -85,B 0,C 180,E1 21756.849,E2 21756.849} C_VEL
LIN {X 0,Y 560.255,Z 513.251,A -85,B 0,C 180,E1 21756.282,E2 21756.282} C_VEL
LIN {X 0,Y 560.272,Z 513.251,A -85,B 0,C 180,E1 21752.938,E2 21752.938} C_VEL
LIN {X 0,Y 560.257,Z 513.244,A -85,B 0,C 180,E1 21749.665,E2 21749.665} C_VEL
LIN {X 0,Y 560.275,Z 513.26,A -85,B 0,C 180,E1 21746.266,E2 21746.266} C_VEL
LIN {X 0,Y 560.279,Z 513.249,A -85,B 0,C 180,E1 21742.901,E2 21742.901} C_VEL
LIN {X 0,Y 560.259,Z 513.249,A -85,B 0,C 180,E1 21739.622,E2 21739.622} C_VEL
LIN {X 0,Y 560.275,Z 513.248,A -85,B 0,C 180,E1 21736.283,E2 21736.283} C_VEL
LIN {X 0,Y 560.25,Z 513.244,A -85,B 0,C 180,E1 21732.98,E2 21732.98} C_VEL
LIN {X 0,Y 560.29,Z 513.523,A -85,B 0,C 180,E1 21730.948,E2 21730.948} C_VEL
LIN {X 0,Y 561.634,Z 516.858,A -85,B 0,C 180,E1 21730.52,E2 21730.52} C_VEL
LIN {X 0,Y 567.548,Z 530.101,A -85,B 0,C 180,E1 21729.065,E2 21729.065} C_VEL
LIN {X 0,Y 566.417,Z 577.209,A -85,B 0,C 180,E1 21725.878,E2 21725.878} C_VEL
LIN {X 0,Y 566.24,Z 590.531,A -85,B 0,C 180,E1 21725.029,E2 21725.029} C_VEL
LIN {X 0,Y 567.769,Z 600.034,A -85,B 0,C 180,E1 21724.775,E2 21724.775} C_VEL
LIN {X 0,Y 566.366,Z 829.311,A -85,B 0,C 180,E1 21721.469,E2 21721.469} C_VEL
LIN {X 0,Y 565.937,Z 896.992,A -85,B 0,C 180,E1 21720.479,E2 21720.479} C_VEL
LIN {X 0,Y 565.545,Z 918.438,A -85,B 0,C 180,E1 21719.973,E2 21719.973} C_VEL
LIN {X 0,Y 565.077,Z 940.12,A -85,B 0,C 180,E1 21719.27,E2 21719.27} C_VEL
LIN {X 0,Y 564.595,Z 959.909,A -85,B 0,C 180,E1 21718.449,E2 21718.449} C_VEL
LIN {X 0,Y 563.994,Z 979.465,A -85,B 0,C 180,E1 21717.447,E2 21717.447} C_VEL
LIN {X 0,Y 563.353,Z 1000.191,A -85,B 0,C 180,E1 21716.171,E2 21716.171} C_VEL
LIN {X 0,Y 562.729,Z 1019.076,A -85,B 0,C 180,E1 21714.792,E2 21714.792} C_VEL
LIN {X 0,Y 562.125,Z 1036.91,A -85,B 0,C 180,E1 21713.258,E2 21713.258} C_VEL
LIN {X 0,Y 561.603,Z 1053.262,A -85,B 0,C 180,E1 21711.625,E2 21711.625} C_VEL
LIN {X 0,Y 561.126,Z 1069.166,A -85,B 0,C 180,E1 21709.789,E2 21709.789} C_VEL
LIN {X 0,Y 560.754,Z 1082.82,A -85,B 0,C 180,E1 21707.967,E2 21707.967} C_VEL
LIN {X 0,Y 560.43,Z 1095.696,A -85,B 0,C 180,E1 21705.947,E2 21705.947} C_VEL
LIN {X 0,Y 560.205,Z 1107.091,A -85,B 0,C 180,E1 21703.837,E2 21703.837} C_VEL
LIN {X 0,Y 560.062,Z 1116.577,A -85,B 0,C 180,E1 21701.743,E2 21701.743} C_VEL
LIN {X 0,Y 559.974,Z 1124.01,A -85,B 0,C 180,E1 21699.727,E2 21699.727} C_VEL
LIN {X 0,Y 559.922,Z 1130.534,A -85,B 0,C 180,E1 21697.49,E2 21697.49} C_VEL
LIN {X 0,Y 559.913,Z 1135.044,A -85,B 0,C 180,E1 21695.431,E2 21695.431} C_VEL
LIN {X 0,Y 559.912,Z 1138.123,A -85,B 0,C 180,E1 21693.276,E2 21693.276} C_VEL
LIN {X 0,Y 559.91,Z 1139.773,A -85,B 0,C 180,E1 21691.023,E2 21691.023} C_VEL
LIN {X 0,Y 559.912,Z 1139.77,A -85,B 0,C 180,E1 21688.874,E2 21688.874} C_VEL
LIN {X 0,Y 559.915,Z 1138.11,A -85,B 0,C 180,E1 21686.622,E2 21686.622} C_VEL
LIN {X 0,Y 559.915,Z 1135.017,A -85,B 0,C 180,E1 21684.466,E2 21684.466} C_VEL
LIN {X 0,Y 559.923,Z 1130.501,A -85,B 0,C 180,E1 21682.407,E2 21682.407} C_VEL
LIN {X 0,Y 559.976,Z 1123.829,A -85,B 0,C 180,E1 21680.13,E2 21680.13} C_VEL
LIN {X 0,Y 560.073,Z 1116.096,A -85,B 0,C 180,E1 21678.044,E2 21678.044} C_VEL
LIN {X 0,Y 560.22,Z 1106.496,A -85,B 0,C 180,E1 21675.952,E2 21675.952} C_VEL
LIN {X 0,Y 560.449,Z 1094.962,A -85,B 0,C 180,E1 21673.841,E2 21673.841} C_VEL
LIN {X 0,Y 560.763,Z 1082.307,A -85,B 0,C 180,E1 21671.871,E2 21671.871} C_VEL
LIN {X 0,Y 561.158,Z 1068.169,A -85,B 0,C 180,E1 21669.995,E2 21669.995} C_VEL
LIN {X 0,Y 561.609,Z 1053.084,A -85,B 0,C 180,E1 21668.265,E2 21668.265} C_VEL
LIN {X 0,Y 562.143,Z 1036.392,A -85,B 0,C 180,E1 21666.605,E2 21666.605} C_VEL
LIN {X 0,Y 562.738,Z 1018.811,A -85,B 0,C 180,E1 21665.096,E2 21665.096} C_VEL
LIN {X 0,Y 563.369,Z 999.777,A -85,B 0,C 180,E1 21663.711,E2 21663.711} C_VEL
LIN {X 0,Y 563.976,Z 980.037,A -85,B 0,C 180,E1 21662.494,E2 21662.494} C_VEL
LIN {X 0,Y 564.583,Z 960.497,A -85,B 0,C 180,E1 21661.486,E2 21661.486} C_VEL
LIN {X 0,Y 565.097,Z 939.65,A -85,B 0,C 180,E1 21660.623,E2 21660.623} C_VEL
LIN {X 0,Y 565.557,Z 917.278,A -85,B 0,C 180,E1 21659.905,E2 21659.905} C_VEL
LIN {X 0,Y 565.948,Z 895.728,A -85,B 0,C 180,E1 21659.41,E2 21659.41} C_VEL
LIN {X 0,Y 567.272,Z 675.248,A -85,B 0,C 180,E1 21656.229,E2 21656.229} C_VEL
LIN {X 0,Y 567.541,Z 599.846,A -85,B 0,C 180,E1 21655.116,E2 21655.116} C_VEL
LIN {X 0,Y 565.599,Z 590.557,A -85,B 0,C 180,E1 21654.809,E2 21654.809} C_VEL
LIN {X 0,Y 566.602,Z 549.997,A -85,B 0,C 180,E1 21651.541,E2 21651.541} C_VEL
LIN {X 0,Y 567.017,Z 529.878,A -85,B 0,C 180,E1 21649.856,E2 21649.856} C_VEL
LIN {X 0,Y 561.228,Z 516.248,A -85,B 0,C 180,E1 21648.133,E2 21648.133} C_VEL
LIN {X 0,Y 560.294,Z 513.449,A -85,B 0,C 180,E1 21647.734,E2 21647.734} C_VEL
LIN {X 0,Y 560.218,Z 513.261,A -85,B 0,C 180,E1 21644.446,E2 21644.446} C_VEL
LIN {X 0,Y 560.276,Z 513.235,A -85,B 0,C 180,E1 21641.296,E2 21641.296} C_VEL
LIN {X 0,Y 560.214,Z 513.259,A -85,B 0,C 180,E1 21638.085,E2 21638.085} C_VEL
LIN {X 0,Y 560.312,Z 513.495,A -85,B 0,C 180,E1 21634.954,E2 21634.954} C_VEL
LIN {X 0,Y 564.132,Z 525.548,A -85,B 0,C 180,E1 21633.772,E2 21633.772} C_VEL
LIN {X 0,Y 563.923,Z 559.268,A -85,B 0,C 180,E1 21631.18,E2 21631.18} C_VEL
LIN {X 0,Y 563.564,Z 595.992,A -85,B 0,C 180,E1 21628.358,E2 21628.358} C_VEL
LIN {X 0,Y 562.783,Z 638.302,A -85,B 0,C 180,E1 21625.084,E2 21625.084} C_VEL
LIN {X 0,Y 562.087,Z 679.907,A -85,B 0,C 180,E1 21621.935,E2 21621.935} C_VEL
LIN {X 0,Y 561.778,Z 705.595,A -85,B 0,C 180,E1 21620.049,E2 21620.049} C_VEL
LIN {X 0,Y 562.512,Z 713.166,A -85,B 0,C 180,E1 21619.919,E2 21619.919} C_VEL
LIN {X 0,Y 561.981,Z 876.026,A -85,B 0,C 180,E1 21617.756,E2 21617.756} C_VEL
LIN {X 0,Y 561.792,Z 893.642,A -85,B 0,C 180,E1 21617.321,E2 21617.321} C_VEL
LIN {X 0,Y 561.542,Z 911.403,A -85,B 0,C 180,E1 21616.675,E2 21616.675} C_VEL
LIN {X 0,Y 561.283,Z 927.408,A -85,B 0,C 180,E1 21615.887,E2 21615.887} C_VEL
LIN {X 0,Y 561.001,Z 942.7,A -85,B 0,C 180,E1 21614.924,E2 21614.924} C_VEL
LIN {X 0,Y 560.707,Z 957.953,A -85,B 0,C 180,E1 21613.72,E2 21613.72} C_VEL
LIN {X 0,Y 560.465,Z 970.816,A -85,B 0,C 180,E1 21612.466,E2 21612.466} C_VEL
LIN {X 0,Y 560.272,Z 982.203,A -85,B 0,C 180,E1 21611.113,E2 21611.113} C_VEL
LIN {X 0,Y 560.116,Z 992.862,A -85,B 0,C 180,E1 21609.556,E2 21609.556} C_VEL
LIN {X 0,Y 560.011,Z 1001.866,A -85,B 0,C 180,E1 21607.902,E2 21607.902} C_VEL
LIN {X 0,Y 559.953,Z 1008.815,A -85,B 0,C 180,E1 21606.253,E2 21606.253} C_VEL
LIN {X 0,Y 559.923,Z 1014.223,A -85,B 0,C 180,E1 21604.507,E2 21604.507} C_VEL
LIN {X 0,Y 559.914,Z 1017.963,A -85,B 0,C 180,E1 21602.661,E2 21602.661} C_VEL
LIN {X 0,Y 559.914,Z 1019.782,A -85,B 0,C 180,E1 21600.819,E2 21600.819} C_VEL
LIN {X 0,Y 559.915,Z 1019.754,A -85,B 0,C 180,E1 21599.079,E2 21599.079} C_VEL
LIN {X 0,Y 559.914,Z 1018.102,A -85,B 0,C 180,E1 21597.339,E2 21597.339} C_VEL
LIN {X 0,Y 559.924,Z 1014.45,A -85,B 0,C 180,E1 21595.494,E2 21595.494} C_VEL
LIN {X 0,Y 559.947,Z 1009.467,A -85,B 0,C 180,E1 21593.85,E2 21593.85} C_VEL
LIN {X 0,Y 560.002,Z 1002.79,A -85,B 0,C 180,E1 21592.202,E2 21592.202} C_VEL
LIN {X 0,Y 560.1,Z 994.051,A -85,B 0,C 180,E1 21590.548,E2 21590.548} C_VEL
LIN {X 0,Y 560.249,Z 983.602,A -85,B 0,C 180,E1 21588.984,E2 21588.984} C_VEL
LIN {X 0,Y 560.457,Z 971.133,A -85,B 0,C 180,E1 21587.482,E2 21587.482} C_VEL
LIN {X 0,Y 560.682,Z 958.912,A -85,B 0,C 180,E1 21586.28,E2 21586.28} C_VEL
LIN {X 0,Y 560.966,Z 944.684,A -85,B 0,C 180,E1 21585.128,E2 21585.128} C_VEL
LIN {X 0,Y 561.236,Z 929.209,A -85,B 0,C 180,E1 21584.13,E2 21584.13} C_VEL
LIN {X 0,Y 561.477,Z 914.858,A -85,B 0,C 180,E1 21583.393,E2 21583.393} C_VEL
LIN {X 0,Y 561.753,Z 898.291,A -85,B 0,C 180,E1 21582.734,E2 21582.734} C_VEL
LIN {X 0,Y 561.939,Z 881.224,A -85,B 0,C 180,E1 21582.263,E2 21582.263} C_VEL
LIN {X 0,Y 562.041,Z 859.691,A -85,B 0,C 180,E1 21581.913,E2 21581.913} C_VEL
LIN {X 0,Y 562.34,Z 709.562,A -85,B 0,C 180,E1 21579.937,E2 21579.937} C_VEL
LIN {X 0,Y 561.724,Z 704.581,A -85,B 0,C 180,E1 21579.812,E2 21579.812} C_VEL
LIN {X 0,Y 562.431,Z 660.74,A -85,B 0,C 180,E1 21576.534,E2 21576.534} C_VEL
LIN {X 0,Y 563.168,Z 616.369,A -85,B 0,C 180,E1 21573.138,E2 21573.138} C_VEL
LIN {X 0,Y 563.655,Z 583.917,A -85,B 0,C 180,E1 21570.628,E2 21570.628} C_VEL
LIN {X 0,Y 563.491,Z 547.039,A -85,B 0,C 180,E1 21568.013,E2 21568.013} C_VEL
LIN {X 0,Y 562.8,Z 523.102,A -85,B 0,C 180,E1 21566.431,E2 21566.431} C_VEL
LIN {X 0,Y 560.29,Z 513.612,A -85,B 0,C 180,E1 21565.735,E2 21565.735} C_VEL
LIN {X 0,Y 560.282,Z 513.261,A -85,B 0,C 180,E1 21565.301,E2 21565.301} C_VEL
LIN {X 0,Y 560.244,Z 513.261,A -85,B 0,C 180,E1 21561.997,E2 21561.997} C_VEL
LIN {X 0,Y 560.28,Z 513.25,A -85,B 0,C 180,E1 21558.678,E2 21558.678} C_VEL
LIN {X 0,Y 560.263,Z 513.242,A -85,B 0,C 180,E1 21555.321,E2 21555.321} C_VEL
LIN {X 0,Y 560.314,Z 513.497,A -85,B 0,C 180,E1 21553.722,E2 21553.722} C_VEL
LIN {X 0,Y 561.83,Z 517.123,A -85,B 0,C 180,E1 21553.225,E2 21553.225} C_VEL
LIN {X 0,Y 567.986,Z 531.11,A -85,B 0,C 180,E1 21551.494,E2 21551.494} C_VEL
LIN {X 0,Y 567.775,Z 543.823,A -85,B 0,C 180,E1 21550.521,E2 21550.521} C_VEL
LIN {X 0,Y 570.247,Z 555.486,A -85,B 0,C 180,E1 21550.113,E2 21550.113} C_VEL
LIN {X 0,Y 568.737,Z 763.338,A -85,B 0,C 180,E1 21546.952,E2 21546.952} C_VEL
LIN {X 0,Y 567.809,Z 891.976,A -85,B 0,C 180,E1 21545.018,E2 21545.018} C_VEL
LIN {X 0,Y 567.323,Z 915.748,A -85,B 0,C 180,E1 21544.473,E2 21544.473} C_VEL
LIN {X 0,Y 566.85,Z 937.735,A -85,B 0,C 180,E1 21543.78,E2 21543.78} C_VEL
LIN {X 0,Y 566.166,Z 959.683,A -85,B 0,C 180,E1 21542.892,E2 21542.892} C_VEL
LIN {X 0,Y 565.506,Z 980.784,A -85,B 0,C 180,E1 21541.855,E2 21541.855} C_VEL
LIN {X 0,Y 564.723,Z 1001.844,A -85,B 0,C 180,E1 21540.605,E2 21540.605} C_VEL
LIN {X 0,Y 563.96,Z 1022.403,A -85,B 0,C 180,E1 21539.18,E2 21539.18} C_VEL
LIN {X 0,Y 563.25,Z 1040.587,A -85,B 0,C 180,E1 21537.716,E2 21537.716} C_VEL
LIN {X 0,Y 562.524,Z 1059.962,A -85,B 0,C 180,E1 21535.923,E2 21535.923} C_VEL
LIN {X 0,Y 561.909,Z 1077.16,A -85,B 0,C 180,E1 21534.102,E2 21534.102} C_VEL
LIN {X 0,Y 561.359,Z 1093.098,A -85,B 0,C 180,E1 21532.152,E2 21532.152} C_VEL
LIN {X 0,Y 560.903,Z 1108.335,A -85,B 0,C 180,E1 21530.015,E2 21530.015} C_VEL
